// Nodes/Code Reading/Node_F_VN_ReadPharmaCodeExp2
{attribute 'linkalways'} 
{attribute 'no_explicit_call' := 'This FB is a CLASS and must be accessed using methods or properties'}
{attribute 'enable_dynamic_creation'}
FUNCTION_BLOCK Node_F_VN_ReadPharmaCodeExp2 EXTENDS VisionNode
VAR
    ipSrcImage : _ITcVnImage;
    ipDecodedData : _ITcVnContainer;
	ipContours : _ITcVnContainer;
	nCodeNumber : _DINT(1);
	nMinBarNumber : _INT(4);
	ipAngles : _ITcVnContainer;
    hrPrev : _HRESULT(S_OK);
	hresult : _HRESULT(S_OK);
END_VAR

METHOD FB_init : BOOL
VAR_INPUT
	bInitRetains : BOOL; // if TRUE, the retain variables are initialized (warm start / cold start)
	bInCopyCode : BOOL;  // if TRUE, the instance afterwards gets moved into the copy code (online change)
END_VAR
AddInput('ipSrcImage', ipSrcImage);
AddInput('hrPrev', hrPrev);
AddParameter('nCodeNumber',nCodeNumber);
AddParameter('nMinBarNumber',nMinBarNumber);
AddOutput('ipDecodedData', ipDecodedData);
AddOutput('ipContours', ipDecodedData);
AddOutput('ipAngles', ipAngles);
AddOutput('hresult',hresult);
END_METHOD

METHOD PUBLIC  Clone : I_Node
VAR
	pNode : POINTER TO Node_F_VN_ReadPharmaCodeExp2;
END_VAR
pNode := __NEW(Node_F_VN_ReadPharmaCodeExp2);
Clone := pNode^;
END_METHOD

METHOD PROTECTED OnExecute
hresult.Value := F_VN_ReadPharmaCodeExp2(
	ipSrcImage := ipSrcImage.Value,
    ipDecodedData := ipDecodedData.Value,
	ipContours := ipContours.Value,
	nCodeNumber := nCodeNumber.Value,
	nMinBarNumber := nMinBarNumber.Value,
	ipAngles := ipAngles.Value,
	hrPrev:= hrPrev.Value);
END_METHOD

METHOD PUBLIC PreExecutionCheck
VAR_INPUT
	Check : I_PreExecutionChecks;
END_VAR
Check.IsTrue(ipSrcImage.IsValid, 'ipSrcImage must contain an image');
Check.IsTrue((ipSrcImage.HasChannelCount(1) OR ipSrcImage.HasChannelCount(3)), 'ipSrcImage must have 1 or 3 channels');

IF (ipSrcImage.HasChannelCount(1)) THEN
    Check.IsTrue(ipSrcImage.IsPixelDepth(8), 'ipSrcImage must have 8 bit pixel depth');
END_IF

IF (ipSrcImage.HasChannelCount(3)) THEN
    Check.IsTrue((ipSrcImage.IsPixelDepth(8) OR 
                 ipSrcImage.IsPixelDepth(16) OR
                 ipSrcImage.IsPixelDepth(32)), 'ipSrcImage must have 8, 16 or 32 bit pixel depth');
END_IF

Check.IsTrue((nCodeNumber.Value = 1), 'nCodeNumber, currently only 1 supported');
END_METHOD

END_FUNCTION_BLOCK

// Nodes/Code Reading/Node_F_VN_ReadQRCode
{attribute 'linkalways'} 
{attribute 'no_explicit_call' := 'This FB is a CLASS and must be accessed using methods or properties'}
{attribute 'enable_dynamic_creation'}
FUNCTION_BLOCK Node_F_VN_ReadQRCode EXTENDS VisionNode
VAR
    ipSrcImage : _ITcVnImage;
    ipDecodedData : _ITcVnContainer;
    hrPrev : _HRESULT(S_OK);
	hresult : _HRESULT(S_OK);
END_VAR

METHOD FB_init : BOOL
VAR_INPUT
	bInitRetains : BOOL; // if TRUE, the retain variables are initialized (warm start / cold start)
	bInCopyCode : BOOL;  // if TRUE, the instance afterwards gets moved into the copy code (online change)
END_VAR
AddInput('ipSrcImage', ipSrcImage);
AddInput('hrPrev', hrPrev);
AddOutput('ipDecodedData', ipDecodedData);
AddOutput('hresult',hresult);
END_METHOD

METHOD PUBLIC  Clone : I_Node
VAR
	pNode : POINTER TO Node_F_VN_ReadQRCode;
END_VAR
pNode := __NEW(Node_F_VN_ReadQRCode);
Clone := pNode^;
END_METHOD

METHOD PROTECTED OnExecute
hresult.Value := F_VN_ReadQRCode(
	ipSrcImage := ipSrcImage.Value,
    ipDecodedData := ipDecodedData.Value,
	hrPrev:= hrPrev.Value);
END_METHOD

METHOD PUBLIC PreExecutionCheck
VAR_INPUT
	Check : I_PreExecutionChecks;
END_VAR
Check.IsTrue(ipSrcImage.IsValid, 'ipSrcImage must contain an image');
Check.IsTrue((ipSrcImage.HasChannelCount(1) OR ipSrcImage.HasChannelCount(3)), 'ipSrcImage must have 1 or 3 channels');
Check.IsTrue(ipSrcImage.IsPixelDepth(8), 'ipSrcImage must have 8 bit pixel depth');
END_METHOD

END_FUNCTION_BLOCK

// Nodes/Code Reading/Node_F_VN_ReadQRCodeExp
{attribute 'linkalways'} 
{attribute 'no_explicit_call' := 'This FB is a CLASS and must be accessed using methods or properties'}
{attribute 'enable_dynamic_creation'}
FUNCTION_BLOCK Node_F_VN_ReadQRCodeExp EXTENDS VisionNode
VAR
    ipSrcImage : _ITcVnImage;
    ipDecodedData : _ITcVnContainer;
	ipContours : _ITcVnContainer;
	nCodeNumber : _DINT(1);
	eSearchStrategy : _UDINT(ETcVn2dCodeSearchStrategy.TCVN_CSS_DEFAULT);
    hrPrev : _HRESULT(S_OK);
	hresult : _HRESULT(S_OK);
END_VAR

METHOD FB_init : BOOL
VAR_INPUT
	bInitRetains : BOOL; // if TRUE, the retain variables are initialized (warm start / cold start)
	bInCopyCode : BOOL;  // if TRUE, the instance afterwards gets moved into the copy code (online change)
END_VAR
AddInput('ipSrcImage', ipSrcImage);
AddInput('hrPrev', hrPrev);
AddParameter('nCodeNumber',nCodeNumber);
AddParameter('eSearchStrategy',eSearchStrategy);
AddOutput('ipDecodedData', ipDecodedData);
AddOutput('ipContours', ipContours);
AddOutput('hresult',hresult);
END_METHOD

METHOD PUBLIC  Clone : I_Node
VAR
	pNode : POINTER TO Node_F_VN_ReadQRCodeExp;
END_VAR
pNode := __NEW(Node_F_VN_ReadQRCodeExp);
Clone := pNode^;
END_METHOD

METHOD PROTECTED OnExecute
hresult.Value := F_VN_ReadQRCodeExp(
	ipSrcImage := ipSrcImage.Value,
    ipDecodedData := ipDecodedData.Value,
	ipContours := ipContours.Value,
	nCodeNumber := nCodeNumber.Value,
	eSearchStrategy := eSearchStrategy.Value,
	hrPrev:= hrPrev.Value);
END_METHOD

METHOD PUBLIC PreExecutionCheck
VAR_INPUT
	Check : I_PreExecutionChecks;
END_VAR
Check.IsTrue(ipSrcImage.IsValid, 'ipSrcImage must contain an image');
Check.IsTrue((ipSrcImage.HasChannelCount(1) OR ipSrcImage.HasChannelCount(3)), 'ipSrcImage must have 1 or 3 channels');
Check.IsTrue(ipSrcImage.IsPixelDepth(8), 'ipSrcImage must have 8 bit pixel depth');
Check.IsTrue((nCodeNumber.Value = 1), 'nCodeNumber, currently only 1 supported');
END_METHOD

END_FUNCTION_BLOCK

// Nodes/Code Reading/Node_F_VN_ReadQRCodeExp2
{attribute 'linkalways'} 
{attribute 'no_explicit_call' := 'This FB is a CLASS and must be accessed using methods or properties'}
{attribute 'enable_dynamic_creation'}
FUNCTION_BLOCK Node_F_VN_ReadQRCodeExp2 EXTENDS VisionNode
VAR
    ipSrcImage : _ITcVnImage;
    ipDecodedData : _ITcVnContainer;
	ipContours : _ITcVnContainer;
	nCodeNumber : _DINT(1);
	eSearchStrategy : _UDINT(ETcVn2dCodeSearchStrategy.TCVN_CSS_DEFAULT);
	ipAngles : _ITcVnContainer;
    hrPrev : _HRESULT(S_OK);
	hresult : _HRESULT(S_OK);
END_VAR

METHOD FB_init : BOOL
VAR_INPUT
	bInitRetains : BOOL; // if TRUE, the retain variables are initialized (warm start / cold start)
	bInCopyCode : BOOL;  // if TRUE, the instance afterwards gets moved into the copy code (online change)
END_VAR
AddInput('ipSrcImage', ipSrcImage);
AddInput('hrPrev', hrPrev);
AddParameter('nCodeNumber',nCodeNumber);
AddParameter('eSearchStrategy',eSearchStrategy);
AddOutput('ipDecodedData', ipDecodedData);
AddOutput('ipContours', ipContours);
AddOutput('ipAngles', ipAngles);
AddOutput('hresult',hresult);
END_METHOD

METHOD PUBLIC  Clone : I_Node
VAR
	pNode : POINTER TO Node_F_VN_ReadQRCodeExp2;
END_VAR
pNode := __NEW(Node_F_VN_ReadQRCodeExp2);
Clone := pNode^;
END_METHOD

METHOD PROTECTED OnExecute
hresult.Value := F_VN_ReadQRCodeExp2(
	ipSrcImage := ipSrcImage.Value,
    ipDecodedData := ipDecodedData.Value,
	ipContours := ipContours.Value,
	nCodeNumber := nCodeNumber.Value,
	eSearchStrategy := eSearchStrategy.Value,
	ipAngles := ipAngles.Value,
	hrPrev:= hrPrev.Value);
END_METHOD

METHOD PUBLIC PreExecutionCheck
VAR_INPUT
	Check : I_PreExecutionChecks;
END_VAR
Check.IsTrue(ipSrcImage.IsValid, 'ipSrcImage must contain an image');
Check.IsTrue((ipSrcImage.HasChannelCount(1) OR ipSrcImage.HasChannelCount(3)), 'ipSrcImage must have 1 or 3 channels');
Check.IsTrue(ipSrcImage.IsPixelDepth(8), 'ipSrcImage must have 8 bit pixel depth');
Check.IsTrue((nCodeNumber.Value = 1), 'nCodeNumber, currently only 1 supported');
END_METHOD

END_FUNCTION_BLOCK

// Nodes/Constants/Node_ContainerType_String_SINT
{attribute 'linkalways'} 
{attribute 'no_explicit_call' := 'This FB is a CLASS and must be accessed using methods or properties'}
{attribute 'enable_dynamic_creation'}
FUNCTION_BLOCK Node_ContainerType_String_SINT EXTENDS Node
VAR
    out : _GUID;
END_VAR

METHOD FB_init : BOOL
VAR_INPUT
	bInitRetains : BOOL; // if TRUE, the retain variables are initialized (warm start / cold start)
	bInCopyCode : BOOL;  // if TRUE, the instance afterwards gets moved into the copy code (online change)
END_VAR
AddOutput('out', out);
END_METHOD

METHOD PUBLIC  Clone : I_Node
VAR
	pNode : POINTER TO Node_ContainerType_String_SINT;
END_VAR
pNode := __NEW(Node_ContainerType_String_SINT);
Clone := pNode^;
END_METHOD

METHOD PROTECTED OnExecute
out.Value := ContainerType_String_SINT;
END_METHOD

END_FUNCTION_BLOCK

// Nodes/Constants/Node_ContainerType_Vector_DINT
{attribute 'linkalways'} 
{attribute 'no_explicit_call' := 'This FB is a CLASS and must be accessed using methods or properties'}
{attribute 'enable_dynamic_creation'}
FUNCTION_BLOCK Node_ContainerType_Vector_DINT EXTENDS Node
VAR
    out : _GUID;
END_VAR

METHOD FB_init : BOOL
VAR_INPUT
	bInitRetains : BOOL; // if TRUE, the retain variables are initialized (warm start / cold start)
	bInCopyCode : BOOL;  // if TRUE, the instance afterwards gets moved into the copy code (online change)
END_VAR
AddOutput('out', out);
END_METHOD

METHOD PUBLIC  Clone : I_Node
VAR
	pNode : POINTER TO Node_ContainerType_Vector_DINT;
END_VAR
pNode := __NEW(Node_ContainerType_Vector_DINT);
Clone := pNode^;
END_METHOD

METHOD PROTECTED OnExecute
out.Value := ContainerType_Vector_DINT;
END_METHOD

END_FUNCTION_BLOCK

// Nodes/Constants/Node_ContainerType_Vector_INT
{attribute 'linkalways'} 
{attribute 'no_explicit_call' := 'This FB is a CLASS and must be accessed using methods or properties'}
{attribute 'enable_dynamic_creation'}
FUNCTION_BLOCK Node_ContainerType_Vector_INT EXTENDS Node
VAR
    out : _GUID;
END_VAR

METHOD FB_init : BOOL
VAR_INPUT
	bInitRetains : BOOL; // if TRUE, the retain variables are initialized (warm start / cold start)
	bInCopyCode : BOOL;  // if TRUE, the instance afterwards gets moved into the copy code (online change)
END_VAR
AddOutput('out', out);
END_METHOD

METHOD PUBLIC  Clone : I_Node
VAR
	pNode : POINTER TO Node_ContainerType_Vector_INT;
END_VAR
pNode := __NEW(Node_ContainerType_Vector_INT);
Clone := pNode^;
END_METHOD

METHOD PROTECTED OnExecute
out.Value := ContainerType_Vector_INT;
END_METHOD

END_FUNCTION_BLOCK

// Nodes/Constants/Node_ContainerType_Vector_ITcVnImage
{attribute 'linkalways'} 
{attribute 'no_explicit_call' := 'This FB is a CLASS and must be accessed using methods or properties'}
{attribute 'enable_dynamic_creation'}
FUNCTION_BLOCK Node_ContainerType_Vector_ITcVnImage EXTENDS Node
VAR
    out : _GUID;
END_VAR

METHOD FB_init : BOOL
VAR_INPUT
	bInitRetains : BOOL; // if TRUE, the retain variables are initialized (warm start / cold start)
	bInCopyCode : BOOL;  // if TRUE, the instance afterwards gets moved into the copy code (online change)
END_VAR
AddOutput('out', out);
END_METHOD

METHOD PUBLIC  Clone : I_Node
VAR
	pNode : POINTER TO Node_ContainerType_Vector_ITcVnImage;
END_VAR
pNode := __NEW(Node_ContainerType_Vector_ITcVnImage);
Clone := pNode^;
END_METHOD

METHOD PROTECTED OnExecute
out.Value := ContainerType_Vector_ITcVnImage;
END_METHOD

END_FUNCTION_BLOCK

// Nodes/Constants/Node_ContainerType_Vector_LREAL
{attribute 'linkalways'} 
{attribute 'no_explicit_call' := 'This FB is a CLASS and must be accessed using methods or properties'}
{attribute 'enable_dynamic_creation'}
FUNCTION_BLOCK Node_ContainerType_Vector_LREAL EXTENDS Node
VAR
    out : _GUID;
END_VAR

METHOD FB_init : BOOL
VAR_INPUT
	bInitRetains : BOOL; // if TRUE, the retain variables are initialized (warm start / cold start)
	bInCopyCode : BOOL;  // if TRUE, the instance afterwards gets moved into the copy code (online change)
END_VAR
AddOutput('out', out);
END_METHOD

METHOD PUBLIC  Clone : I_Node
VAR
	pNode : POINTER TO Node_ContainerType_Vector_LREAL;
END_VAR
pNode := __NEW(Node_ContainerType_Vector_LREAL);
Clone := pNode^;
END_METHOD

METHOD PROTECTED OnExecute
out.Value := ContainerType_Vector_LREAL;
END_METHOD

END_FUNCTION_BLOCK

// Nodes/Constants/Node_ContainerType_Vector_REAL
{attribute 'linkalways'} 
{attribute 'no_explicit_call' := 'This FB is a CLASS and must be accessed using methods or properties'}
{attribute 'enable_dynamic_creation'}
FUNCTION_BLOCK Node_ContainerType_Vector_REAL EXTENDS Node
VAR
    out : _GUID;
END_VAR

METHOD FB_init : BOOL
VAR_INPUT
	bInitRetains : BOOL; // if TRUE, the retain variables are initialized (warm start / cold start)
	bInCopyCode : BOOL;  // if TRUE, the instance afterwards gets moved into the copy code (online change)
END_VAR
AddOutput('out', out);
END_METHOD

METHOD PUBLIC  Clone : I_Node
VAR
	pNode : POINTER TO Node_ContainerType_Vector_REAL;
END_VAR
pNode := __NEW(Node_ContainerType_Vector_REAL);
Clone := pNode^;
END_METHOD

METHOD PROTECTED OnExecute
out.Value := ContainerType_Vector_REAL;
END_METHOD

END_FUNCTION_BLOCK

// Nodes/Constants/Node_ContainerType_Vector_SINT
{attribute 'linkalways'} 
{attribute 'no_explicit_call' := 'This FB is a CLASS and must be accessed using methods or properties'}
{attribute 'enable_dynamic_creation'}
FUNCTION_BLOCK Node_ContainerType_Vector_SINT EXTENDS Node
VAR
    out : _GUID;
END_VAR

METHOD FB_init : BOOL
VAR_INPUT
	bInitRetains : BOOL; // if TRUE, the retain variables are initialized (warm start / cold start)
	bInCopyCode : BOOL;  // if TRUE, the instance afterwards gets moved into the copy code (online change)
END_VAR
AddOutput('out', out);
END_METHOD

METHOD PUBLIC  Clone : I_Node
VAR
	pNode : POINTER TO Node_ContainerType_Vector_SINT;
END_VAR
pNode := __NEW(Node_ContainerType_Vector_SINT);
Clone := pNode^;
END_METHOD

METHOD PROTECTED OnExecute
out.Value := ContainerType_Vector_SINT;
END_METHOD

END_FUNCTION_BLOCK

// Nodes/Constants/Node_ContainerType_Vector_String_SINT
{attribute 'linkalways'} 
{attribute 'no_explicit_call' := 'This FB is a CLASS and must be accessed using methods or properties'}
{attribute 'enable_dynamic_creation'}
FUNCTION_BLOCK Node_ContainerType_Vector_String_SINT EXTENDS Node
VAR
    out : _GUID;
END_VAR

METHOD FB_init : BOOL
VAR_INPUT
	bInitRetains : BOOL; // if TRUE, the retain variables are initialized (warm start / cold start)
	bInCopyCode : BOOL;  // if TRUE, the instance afterwards gets moved into the copy code (online change)
END_VAR
AddOutput('out', out);
END_METHOD

METHOD PUBLIC  Clone : I_Node
VAR
	pNode : POINTER TO Node_ContainerType_Vector_String_SINT;
END_VAR
pNode := __NEW(Node_ContainerType_Vector_String_SINT);
Clone := pNode^;
END_METHOD

METHOD PROTECTED OnExecute
out.Value := ContainerType_Vector_String_SINT;
END_METHOD

END_FUNCTION_BLOCK

// Nodes/Constants/Node_ContainerType_Vector_TcVnDMatch
{attribute 'linkalways'} 
{attribute 'no_explicit_call' := 'This FB is a CLASS and must be accessed using methods or properties'}
{attribute 'enable_dynamic_creation'}
FUNCTION_BLOCK Node_ContainerType_Vector_TcVnDMatch EXTENDS Node
VAR
    out : _GUID;
END_VAR

METHOD FB_init : BOOL
VAR_INPUT
	bInitRetains : BOOL; // if TRUE, the retain variables are initialized (warm start / cold start)
	bInCopyCode : BOOL;  // if TRUE, the instance afterwards gets moved into the copy code (online change)
END_VAR
AddOutput('out', out);
END_METHOD

METHOD PUBLIC  Clone : I_Node
VAR
	pNode : POINTER TO Node_ContainerType_Vector_TcVnDMatch;
END_VAR
pNode := __NEW(Node_ContainerType_Vector_TcVnDMatch);
Clone := pNode^;
END_METHOD

METHOD PROTECTED OnExecute
out.Value := ContainerType_Vector_TcVnDMatch;
END_METHOD

END_FUNCTION_BLOCK

// Nodes/Constants/Node_ContainerType_Vector_TcVnKeyPoint
{attribute 'linkalways'} 
{attribute 'no_explicit_call' := 'This FB is a CLASS and must be accessed using methods or properties'}
{attribute 'enable_dynamic_creation'}
FUNCTION_BLOCK Node_ContainerType_Vector_TcVnKeyPoint EXTENDS Node
VAR
    out : _GUID;
END_VAR

METHOD FB_init : BOOL
VAR_INPUT
	bInitRetains : BOOL; // if TRUE, the retain variables are initialized (warm start / cold start)
	bInCopyCode : BOOL;  // if TRUE, the instance afterwards gets moved into the copy code (online change)
END_VAR
AddOutput('out', out);
END_METHOD

METHOD PUBLIC  Clone : I_Node
VAR
	pNode : POINTER TO Node_ContainerType_Vector_TcVnKeyPoint;
END_VAR
pNode := __NEW(Node_ContainerType_Vector_TcVnKeyPoint);
Clone := pNode^;
END_METHOD

METHOD PROTECTED OnExecute
out.Value := ContainerType_Vector_TcVnKeyPoint;
END_METHOD

END_FUNCTION_BLOCK

// Nodes/Constants/Node_ContainerType_Vector_TcVnPoint2_DINT
{attribute 'linkalways'} 
{attribute 'no_explicit_call' := 'This FB is a CLASS and must be accessed using methods or properties'}
{attribute 'enable_dynamic_creation'}
FUNCTION_BLOCK Node_ContainerType_Vector_TcVnPoint2_DINT EXTENDS Node
VAR
    out : _GUID;
END_VAR

METHOD FB_init : BOOL
VAR_INPUT
	bInitRetains : BOOL; // if TRUE, the retain variables are initialized (warm start / cold start)
	bInCopyCode : BOOL;  // if TRUE, the instance afterwards gets moved into the copy code (online change)
END_VAR
AddOutput('out', out);
END_METHOD

METHOD PUBLIC  Clone : I_Node
VAR
	pNode : POINTER TO Node_ContainerType_Vector_TcVnPoint2_DINT;
END_VAR
pNode := __NEW(Node_ContainerType_Vector_TcVnPoint2_DINT);
Clone := pNode^;
END_METHOD

METHOD PROTECTED OnExecute
out.Value := ContainerType_Vector_TcVnPoint2_DINT;
END_METHOD

END_FUNCTION_BLOCK

// Nodes/Constants/Node_ContainerType_Vector_TcVnPoint2_LREAL
{attribute 'linkalways'} 
{attribute 'no_explicit_call' := 'This FB is a CLASS and must be accessed using methods or properties'}
{attribute 'enable_dynamic_creation'}
FUNCTION_BLOCK Node_ContainerType_Vector_TcVnPoint2_LREAL EXTENDS Node
VAR
    out : _GUID;
END_VAR

METHOD FB_init : BOOL
VAR_INPUT
	bInitRetains : BOOL; // if TRUE, the retain variables are initialized (warm start / cold start)
	bInCopyCode : BOOL;  // if TRUE, the instance afterwards gets moved into the copy code (online change)
END_VAR
AddOutput('out', out);
END_METHOD

METHOD PUBLIC  Clone : I_Node
VAR
	pNode : POINTER TO Node_ContainerType_Vector_TcVnPoint2_LREAL;
END_VAR
pNode := __NEW(Node_ContainerType_Vector_TcVnPoint2_LREAL);
Clone := pNode^;
END_METHOD

METHOD PROTECTED OnExecute
out.Value := ContainerType_Vector_TcVnPoint2_LREAL;
END_METHOD

END_FUNCTION_BLOCK

// Nodes/Constants/Node_ContainerType_Vector_TcVnPoint2_REAL
{attribute 'linkalways'} 
{attribute 'no_explicit_call' := 'This FB is a CLASS and must be accessed using methods or properties'}
{attribute 'enable_dynamic_creation'}
FUNCTION_BLOCK Node_ContainerType_Vector_TcVnPoint2_REAL EXTENDS Node
VAR
    out : _GUID;
END_VAR

METHOD FB_init : BOOL
VAR_INPUT
	bInitRetains : BOOL; // if TRUE, the retain variables are initialized (warm start / cold start)
	bInCopyCode : BOOL;  // if TRUE, the instance afterwards gets moved into the copy code (online change)
END_VAR
AddOutput('out', out);
END_METHOD

METHOD PUBLIC  Clone : I_Node
VAR
	pNode : POINTER TO Node_ContainerType_Vector_TcVnPoint2_REAL;
END_VAR
pNode := __NEW(Node_ContainerType_Vector_TcVnPoint2_REAL);
Clone := pNode^;
END_METHOD

METHOD PROTECTED OnExecute
out.Value := ContainerType_Vector_TcVnPoint2_REAL;
END_METHOD

END_FUNCTION_BLOCK

// Nodes/Constants/Node_ContainerType_Vector_TcVnPoint3_LREAL
{attribute 'linkalways'} 
{attribute 'no_explicit_call' := 'This FB is a CLASS and must be accessed using methods or properties'}
{attribute 'enable_dynamic_creation'}
FUNCTION_BLOCK Node_ContainerType_Vector_TcVnPoint3_LREAL EXTENDS Node
VAR
    out : _GUID;
END_VAR

METHOD FB_init : BOOL
VAR_INPUT
	bInitRetains : BOOL; // if TRUE, the retain variables are initialized (warm start / cold start)
	bInCopyCode : BOOL;  // if TRUE, the instance afterwards gets moved into the copy code (online change)
END_VAR
AddOutput('out', out);
END_METHOD

METHOD PUBLIC  Clone : I_Node
VAR
	pNode : POINTER TO Node_ContainerType_Vector_TcVnPoint3_LREAL;
END_VAR
pNode := __NEW(Node_ContainerType_Vector_TcVnPoint3_LREAL);
Clone := pNode^;
END_METHOD

METHOD PROTECTED OnExecute
out.Value := ContainerType_Vector_TcVnPoint3_LREAL;
END_METHOD

END_FUNCTION_BLOCK

// Nodes/Constants/Node_ContainerType_Vector_TcVnPoint3_REAL
{attribute 'linkalways'} 
{attribute 'no_explicit_call' := 'This FB is a CLASS and must be accessed using methods or properties'}
{attribute 'enable_dynamic_creation'}
FUNCTION_BLOCK Node_ContainerType_Vector_TcVnPoint3_REAL EXTENDS Node
VAR
    out : _GUID;
END_VAR

METHOD FB_init : BOOL
VAR_INPUT
	bInitRetains : BOOL; // if TRUE, the retain variables are initialized (warm start / cold start)
	bInCopyCode : BOOL;  // if TRUE, the instance afterwards gets moved into the copy code (online change)
END_VAR
AddOutput('out', out);
END_METHOD

METHOD PUBLIC  Clone : I_Node
VAR
	pNode : POINTER TO Node_ContainerType_Vector_TcVnPoint3_REAL;
END_VAR
pNode := __NEW(Node_ContainerType_Vector_TcVnPoint3_REAL);
Clone := pNode^;
END_METHOD

METHOD PROTECTED OnExecute
out.Value := ContainerType_Vector_TcVnPoint3_REAL;
END_METHOD

END_FUNCTION_BLOCK

// Nodes/Constants/Node_ContainerType_Vector_TcVnRectangle_DINT
{attribute 'linkalways'} 
{attribute 'no_explicit_call' := 'This FB is a CLASS and must be accessed using methods or properties'}
{attribute 'enable_dynamic_creation'}
FUNCTION_BLOCK Node_ContainerType_Vector_TcVnRectangle_DINT EXTENDS Node
VAR
    out : _GUID;
END_VAR

METHOD FB_init : BOOL
VAR_INPUT
	bInitRetains : BOOL; // if TRUE, the retain variables are initialized (warm start / cold start)
	bInCopyCode : BOOL;  // if TRUE, the instance afterwards gets moved into the copy code (online change)
END_VAR
AddOutput('out', out);
END_METHOD

METHOD PUBLIC  Clone : I_Node
VAR
	pNode : POINTER TO Node_ContainerType_Vector_TcVnRectangle_DINT;
END_VAR
pNode := __NEW(Node_ContainerType_Vector_TcVnRectangle_DINT);
Clone := pNode^;
END_METHOD

METHOD PROTECTED OnExecute
out.Value := ContainerType_Vector_TcVnRectangle_DINT;
END_METHOD

END_FUNCTION_BLOCK

// Nodes/Constants/Node_ContainerType_Vector_TcVnRotatedRectangle
{attribute 'linkalways'} 
{attribute 'no_explicit_call' := 'This FB is a CLASS and must be accessed using methods or properties'}
{attribute 'enable_dynamic_creation'}
FUNCTION_BLOCK Node_ContainerType_Vector_TcVnRotatedRectangle EXTENDS Node
VAR
    out : _GUID;
END_VAR

METHOD FB_init : BOOL
VAR_INPUT
	bInitRetains : BOOL; // if TRUE, the retain variables are initialized (warm start / cold start)
	bInCopyCode : BOOL;  // if TRUE, the instance afterwards gets moved into the copy code (online change)
END_VAR
AddOutput('out', out);
END_METHOD

METHOD PUBLIC  Clone : I_Node
VAR
	pNode : POINTER TO Node_ContainerType_Vector_TcVnRotatedRectangle;
END_VAR
pNode := __NEW(Node_ContainerType_Vector_TcVnRotatedRectangle);
Clone := pNode^;
END_METHOD

METHOD PROTECTED OnExecute
out.Value := ContainerType_Vector_TcVnRotatedRectangle;
END_METHOD

END_FUNCTION_BLOCK

// Nodes/Constants/Node_ContainerType_Vector_TcVnVector2_DINT
{attribute 'linkalways'} 
{attribute 'no_explicit_call' := 'This FB is a CLASS and must be accessed using methods or properties'}
{attribute 'enable_dynamic_creation'}
FUNCTION_BLOCK Node_ContainerType_Vector_TcVnVector2_DINT EXTENDS Node
VAR
    out : _GUID;
END_VAR

METHOD FB_init : BOOL
VAR_INPUT
	bInitRetains : BOOL; // if TRUE, the retain variables are initialized (warm start / cold start)
	bInCopyCode : BOOL;  // if TRUE, the instance afterwards gets moved into the copy code (online change)
END_VAR
AddOutput('out', out);
END_METHOD

METHOD PUBLIC  Clone : I_Node
VAR
	pNode : POINTER TO Node_ContainerType_Vector_TcVnVector2_DINT;
END_VAR
pNode := __NEW(Node_ContainerType_Vector_TcVnVector2_DINT);
Clone := pNode^;
END_METHOD

METHOD PROTECTED OnExecute
out.Value := ContainerType_Vector_TcVnVector2_DINT;
END_METHOD

END_FUNCTION_BLOCK

// Nodes/Constants/Node_ContainerType_Vector_TcVnVector2_INT
{attribute 'linkalways'} 
{attribute 'no_explicit_call' := 'This FB is a CLASS and must be accessed using methods or properties'}
{attribute 'enable_dynamic_creation'}
FUNCTION_BLOCK Node_ContainerType_Vector_TcVnVector2_INT EXTENDS Node
VAR
    out : _GUID;
END_VAR

METHOD FB_init : BOOL
VAR_INPUT
	bInitRetains : BOOL; // if TRUE, the retain variables are initialized (warm start / cold start)
	bInCopyCode : BOOL;  // if TRUE, the instance afterwards gets moved into the copy code (online change)
END_VAR
AddOutput('out', out);
END_METHOD

METHOD PUBLIC  Clone : I_Node
VAR
	pNode : POINTER TO Node_ContainerType_Vector_TcVnVector2_INT;
END_VAR
pNode := __NEW(Node_ContainerType_Vector_TcVnVector2_INT);
Clone := pNode^;
END_METHOD

METHOD PROTECTED OnExecute
out.Value := ContainerType_Vector_TcVnVector2_INT;
END_METHOD

END_FUNCTION_BLOCK

// Nodes/Constants/Node_ContainerType_Vector_TcVnVector2_REAL
{attribute 'linkalways'} 
{attribute 'no_explicit_call' := 'This FB is a CLASS and must be accessed using methods or properties'}
{attribute 'enable_dynamic_creation'}
FUNCTION_BLOCK Node_ContainerType_Vector_TcVnVector2_REAL EXTENDS Node
VAR
    out : _GUID;
END_VAR

METHOD FB_init : BOOL
VAR_INPUT
	bInitRetains : BOOL; // if TRUE, the retain variables are initialized (warm start / cold start)
	bInCopyCode : BOOL;  // if TRUE, the instance afterwards gets moved into the copy code (online change)
END_VAR
AddOutput('out', out);
END_METHOD

METHOD PUBLIC  Clone : I_Node
VAR
	pNode : POINTER TO Node_ContainerType_Vector_TcVnVector2_REAL;
END_VAR
pNode := __NEW(Node_ContainerType_Vector_TcVnVector2_REAL);
Clone := pNode^;
END_METHOD

METHOD PROTECTED OnExecute
out.Value := ContainerType_Vector_TcVnVector2_REAL;
END_METHOD

END_FUNCTION_BLOCK

// Nodes/Constants/Node_ContainerType_Vector_TcVnVector2_SINT
{attribute 'linkalways'} 
{attribute 'no_explicit_call' := 'This FB is a CLASS and must be accessed using methods or properties'}
{attribute 'enable_dynamic_creation'}
FUNCTION_BLOCK Node_ContainerType_Vector_TcVnVector2_SINT EXTENDS Node
VAR
    out : _GUID;
END_VAR

METHOD FB_init : BOOL
VAR_INPUT
	bInitRetains : BOOL; // if TRUE, the retain variables are initialized (warm start / cold start)
	bInCopyCode : BOOL;  // if TRUE, the instance afterwards gets moved into the copy code (online change)
END_VAR
AddOutput('out', out);
END_METHOD

METHOD PUBLIC  Clone : I_Node
VAR
	pNode : POINTER TO Node_ContainerType_Vector_TcVnVector2_SINT;
END_VAR
pNode := __NEW(Node_ContainerType_Vector_TcVnVector2_SINT);
Clone := pNode^;
END_METHOD

METHOD PROTECTED OnExecute
out.Value := ContainerType_Vector_TcVnVector2_SINT;
END_METHOD

END_FUNCTION_BLOCK

// Nodes/Constants/Node_ContainerType_Vector_TcVnVector2_UINT
{attribute 'linkalways'} 
{attribute 'no_explicit_call' := 'This FB is a CLASS and must be accessed using methods or properties'}
{attribute 'enable_dynamic_creation'}
FUNCTION_BLOCK Node_ContainerType_Vector_TcVnVector2_UINT EXTENDS Node
VAR
    out : _GUID;
END_VAR

METHOD FB_init : BOOL
VAR_INPUT
	bInitRetains : BOOL; // if TRUE, the retain variables are initialized (warm start / cold start)
	bInCopyCode : BOOL;  // if TRUE, the instance afterwards gets moved into the copy code (online change)
END_VAR
AddOutput('out', out);
END_METHOD

METHOD PUBLIC  Clone : I_Node
VAR
	pNode : POINTER TO Node_ContainerType_Vector_TcVnVector2_UINT;
END_VAR
pNode := __NEW(Node_ContainerType_Vector_TcVnVector2_UINT);
Clone := pNode^;
END_METHOD

METHOD PROTECTED OnExecute
out.Value := ContainerType_Vector_TcVnVector2_UINT;
END_METHOD

END_FUNCTION_BLOCK

// Nodes/Constants/Node_ContainerType_Vector_TcVnVector2_USINT
{attribute 'linkalways'} 
{attribute 'no_explicit_call' := 'This FB is a CLASS and must be accessed using methods or properties'}
{attribute 'enable_dynamic_creation'}
FUNCTION_BLOCK Node_ContainerType_Vector_TcVnVector2_USINT EXTENDS Node
VAR
    out : _GUID;
END_VAR

METHOD FB_init : BOOL
VAR_INPUT
	bInitRetains : BOOL; // if TRUE, the retain variables are initialized (warm start / cold start)
	bInCopyCode : BOOL;  // if TRUE, the instance afterwards gets moved into the copy code (online change)
END_VAR
AddOutput('out', out);
END_METHOD

METHOD PUBLIC  Clone : I_Node
VAR
	pNode : POINTER TO Node_ContainerType_Vector_TcVnVector2_USINT;
END_VAR
pNode := __NEW(Node_ContainerType_Vector_TcVnVector2_USINT);
Clone := pNode^;
END_METHOD

METHOD PROTECTED OnExecute
out.Value := ContainerType_Vector_TcVnVector2_USINT;
END_METHOD

END_FUNCTION_BLOCK

// Nodes/Constants/Node_ContainerType_Vector_TcVnVector3_INT
{attribute 'linkalways'} 
{attribute 'no_explicit_call' := 'This FB is a CLASS and must be accessed using methods or properties'}
{attribute 'enable_dynamic_creation'}
FUNCTION_BLOCK Node_ContainerType_Vector_TcVnVector3_INT EXTENDS Node
VAR
    out : _GUID;
END_VAR

METHOD FB_init : BOOL
VAR_INPUT
	bInitRetains : BOOL; // if TRUE, the retain variables are initialized (warm start / cold start)
	bInCopyCode : BOOL;  // if TRUE, the instance afterwards gets moved into the copy code (online change)
END_VAR
AddOutput('out', out);
END_METHOD

METHOD PUBLIC  Clone : I_Node
VAR
	pNode : POINTER TO Node_ContainerType_Vector_TcVnVector3_INT;
END_VAR
pNode := __NEW(Node_ContainerType_Vector_TcVnVector3_INT);
Clone := pNode^;
END_METHOD

METHOD PROTECTED OnExecute
out.Value := ContainerType_Vector_TcVnVector3_INT;
END_METHOD

END_FUNCTION_BLOCK

// Nodes/Constants/Node_ContainerType_Vector_TcVnVector3_REAL
{attribute 'linkalways'} 
{attribute 'no_explicit_call' := 'This FB is a CLASS and must be accessed using methods or properties'}
{attribute 'enable_dynamic_creation'}
FUNCTION_BLOCK Node_ContainerType_Vector_TcVnVector3_REAL EXTENDS Node
VAR
    out : _GUID;
END_VAR

METHOD FB_init : BOOL
VAR_INPUT
	bInitRetains : BOOL; // if TRUE, the retain variables are initialized (warm start / cold start)
	bInCopyCode : BOOL;  // if TRUE, the instance afterwards gets moved into the copy code (online change)
END_VAR
AddOutput('out', out);
END_METHOD

METHOD PUBLIC  Clone : I_Node
VAR
	pNode : POINTER TO Node_ContainerType_Vector_TcVnVector3_REAL;
END_VAR
pNode := __NEW(Node_ContainerType_Vector_TcVnVector3_REAL);
Clone := pNode^;
END_METHOD

METHOD PROTECTED OnExecute
out.Value := ContainerType_Vector_TcVnVector3_REAL;
END_METHOD

END_FUNCTION_BLOCK

// Nodes/Constants/Node_ContainerType_Vector_TcVnVector3_SINT
{attribute 'linkalways'} 
{attribute 'no_explicit_call' := 'This FB is a CLASS and must be accessed using methods or properties'}
{attribute 'enable_dynamic_creation'}
FUNCTION_BLOCK Node_ContainerType_Vector_TcVnVector3_SINT EXTENDS Node
VAR
    out : _GUID;
END_VAR

METHOD FB_init : BOOL
VAR_INPUT
	bInitRetains : BOOL; // if TRUE, the retain variables are initialized (warm start / cold start)
	bInCopyCode : BOOL;  // if TRUE, the instance afterwards gets moved into the copy code (online change)
END_VAR
AddOutput('out', out);
END_METHOD

METHOD PUBLIC  Clone : I_Node
VAR
	pNode : POINTER TO Node_ContainerType_Vector_TcVnVector3_SINT;
END_VAR
pNode := __NEW(Node_ContainerType_Vector_TcVnVector3_SINT);
Clone := pNode^;
END_METHOD

METHOD PROTECTED OnExecute
out.Value := ContainerType_Vector_TcVnVector3_SINT;
END_METHOD

END_FUNCTION_BLOCK

// Nodes/Constants/Node_ContainerType_Vector_TcVnVector3_UINT
{attribute 'linkalways'} 
{attribute 'no_explicit_call' := 'This FB is a CLASS and must be accessed using methods or properties'}
{attribute 'enable_dynamic_creation'}
FUNCTION_BLOCK Node_ContainerType_Vector_TcVnVector3_UINT EXTENDS Node
VAR
    out : _GUID;
END_VAR

METHOD FB_init : BOOL
VAR_INPUT
	bInitRetains : BOOL; // if TRUE, the retain variables are initialized (warm start / cold start)
	bInCopyCode : BOOL;  // if TRUE, the instance afterwards gets moved into the copy code (online change)
END_VAR
AddOutput('out', out);
END_METHOD

METHOD PUBLIC  Clone : I_Node
VAR
	pNode : POINTER TO Node_ContainerType_Vector_TcVnVector3_UINT;
END_VAR
pNode := __NEW(Node_ContainerType_Vector_TcVnVector3_UINT);
Clone := pNode^;
END_METHOD

METHOD PROTECTED OnExecute
out.Value := ContainerType_Vector_TcVnVector3_UINT;
END_METHOD

END_FUNCTION_BLOCK

// Nodes/Constants/Node_ContainerType_Vector_TcVnVector3_USINT
{attribute 'linkalways'} 
{attribute 'no_explicit_call' := 'This FB is a CLASS and must be accessed using methods or properties'}
{attribute 'enable_dynamic_creation'}
FUNCTION_BLOCK Node_ContainerType_Vector_TcVnVector3_USINT EXTENDS Node
VAR
    out : _GUID;
END_VAR

METHOD FB_init : BOOL
VAR_INPUT
	bInitRetains : BOOL; // if TRUE, the retain variables are initialized (warm start / cold start)
	bInCopyCode : BOOL;  // if TRUE, the instance afterwards gets moved into the copy code (online change)
END_VAR
AddOutput('out', out);
END_METHOD

METHOD PUBLIC  Clone : I_Node
VAR
	pNode : POINTER TO Node_ContainerType_Vector_TcVnVector3_USINT;
END_VAR
pNode := __NEW(Node_ContainerType_Vector_TcVnVector3_USINT);
Clone := pNode^;
END_METHOD

METHOD PROTECTED OnExecute
out.Value := ContainerType_Vector_TcVnVector3_USINT;
END_METHOD

END_FUNCTION_BLOCK

// Nodes/Constants/Node_ContainerType_Vector_TcVnVector4_DINT
{attribute 'linkalways'} 
{attribute 'no_explicit_call' := 'This FB is a CLASS and must be accessed using methods or properties'}
{attribute 'enable_dynamic_creation'}
FUNCTION_BLOCK Node_ContainerType_Vector_TcVnVector4_DINT EXTENDS Node
VAR
    out : _GUID;
END_VAR

METHOD FB_init : BOOL
VAR_INPUT
	bInitRetains : BOOL; // if TRUE, the retain variables are initialized (warm start / cold start)
	bInCopyCode : BOOL;  // if TRUE, the instance afterwards gets moved into the copy code (online change)
END_VAR
AddOutput('out', out);
END_METHOD

METHOD PUBLIC  Clone : I_Node
VAR
	pNode : POINTER TO Node_ContainerType_Vector_TcVnVector4_DINT;
END_VAR
pNode := __NEW(Node_ContainerType_Vector_TcVnVector4_DINT);
Clone := pNode^;
END_METHOD

METHOD PROTECTED OnExecute
out.Value := ContainerType_Vector_TcVnVector4_DINT;
END_METHOD

END_FUNCTION_BLOCK

// Nodes/Constants/Node_ContainerType_Vector_TcVnVector4_INT
{attribute 'linkalways'} 
{attribute 'no_explicit_call' := 'This FB is a CLASS and must be accessed using methods or properties'}
{attribute 'enable_dynamic_creation'}
FUNCTION_BLOCK Node_ContainerType_Vector_TcVnVector4_INT EXTENDS Node
VAR
    out : _GUID;
END_VAR

METHOD FB_init : BOOL
VAR_INPUT
	bInitRetains : BOOL; // if TRUE, the retain variables are initialized (warm start / cold start)
	bInCopyCode : BOOL;  // if TRUE, the instance afterwards gets moved into the copy code (online change)
END_VAR
AddOutput('out', out);
END_METHOD

METHOD PUBLIC  Clone : I_Node
VAR
	pNode : POINTER TO Node_ContainerType_Vector_TcVnVector4_INT;
END_VAR
pNode := __NEW(Node_ContainerType_Vector_TcVnVector4_INT);
Clone := pNode^;
END_METHOD

METHOD PROTECTED OnExecute
out.Value := ContainerType_Vector_TcVnVector4_INT;
END_METHOD

END_FUNCTION_BLOCK

// Nodes/Constants/Node_ContainerType_Vector_TcVnVector4_LREAL
{attribute 'linkalways'} 
{attribute 'no_explicit_call' := 'This FB is a CLASS and must be accessed using methods or properties'}
{attribute 'enable_dynamic_creation'}
FUNCTION_BLOCK Node_ContainerType_Vector_TcVnVector4_LREAL EXTENDS Node
VAR
    out : _GUID;
END_VAR

METHOD FB_init : BOOL
VAR_INPUT
	bInitRetains : BOOL; // if TRUE, the retain variables are initialized (warm start / cold start)
	bInCopyCode : BOOL;  // if TRUE, the instance afterwards gets moved into the copy code (online change)
END_VAR
AddOutput('out', out);
END_METHOD

METHOD PUBLIC  Clone : I_Node
VAR
	pNode : POINTER TO Node_ContainerType_Vector_TcVnVector4_LREAL;
END_VAR
pNode := __NEW(Node_ContainerType_Vector_TcVnVector4_LREAL);
Clone := pNode^;
END_METHOD

METHOD PROTECTED OnExecute
out.Value := ContainerType_Vector_TcVnVector4_LREAL;
END_METHOD

END_FUNCTION_BLOCK

// Nodes/Constants/Node_ContainerType_Vector_TcVnVector4_REAL
{attribute 'linkalways'} 
{attribute 'no_explicit_call' := 'This FB is a CLASS and must be accessed using methods or properties'}
{attribute 'enable_dynamic_creation'}
FUNCTION_BLOCK Node_ContainerType_Vector_TcVnVector4_REAL EXTENDS Node
VAR
    out : _GUID;
END_VAR

METHOD FB_init : BOOL
VAR_INPUT
	bInitRetains : BOOL; // if TRUE, the retain variables are initialized (warm start / cold start)
	bInCopyCode : BOOL;  // if TRUE, the instance afterwards gets moved into the copy code (online change)
END_VAR
AddOutput('out', out);
END_METHOD

METHOD PUBLIC  Clone : I_Node
VAR
	pNode : POINTER TO Node_ContainerType_Vector_TcVnVector4_REAL;
END_VAR
pNode := __NEW(Node_ContainerType_Vector_TcVnVector4_REAL);
Clone := pNode^;
END_METHOD

METHOD PROTECTED OnExecute
out.Value := ContainerType_Vector_TcVnVector4_REAL;
END_METHOD

END_FUNCTION_BLOCK

// Nodes/Constants/Node_ContainerType_Vector_TcVnVector4_SINT
{attribute 'linkalways'} 
{attribute 'no_explicit_call' := 'This FB is a CLASS and must be accessed using methods or properties'}
{attribute 'enable_dynamic_creation'}
FUNCTION_BLOCK Node_ContainerType_Vector_TcVnVector4_SINT EXTENDS Node
VAR
    out : _GUID;
END_VAR

METHOD FB_init : BOOL
VAR_INPUT
	bInitRetains : BOOL; // if TRUE, the retain variables are initialized (warm start / cold start)
	bInCopyCode : BOOL;  // if TRUE, the instance afterwards gets moved into the copy code (online change)
END_VAR
AddOutput('out', out);
END_METHOD

METHOD PUBLIC  Clone : I_Node
VAR
	pNode : POINTER TO Node_ContainerType_Vector_TcVnVector4_SINT;
END_VAR
pNode := __NEW(Node_ContainerType_Vector_TcVnVector4_SINT);
Clone := pNode^;
END_METHOD

METHOD PROTECTED OnExecute
out.Value := ContainerType_Vector_TcVnVector4_SINT;
END_METHOD

END_FUNCTION_BLOCK

// Nodes/Constants/Node_ContainerType_Vector_TcVnVector4_UINT
{attribute 'linkalways'} 
{attribute 'no_explicit_call' := 'This FB is a CLASS and must be accessed using methods or properties'}
{attribute 'enable_dynamic_creation'}
FUNCTION_BLOCK Node_ContainerType_Vector_TcVnVector4_UINT EXTENDS Node
VAR
    out : _GUID;
END_VAR

METHOD FB_init : BOOL
VAR_INPUT
	bInitRetains : BOOL; // if TRUE, the retain variables are initialized (warm start / cold start)
	bInCopyCode : BOOL;  // if TRUE, the instance afterwards gets moved into the copy code (online change)
END_VAR
AddOutput('out', out);
END_METHOD

METHOD PUBLIC  Clone : I_Node
VAR
	pNode : POINTER TO Node_ContainerType_Vector_TcVnVector4_UINT;
END_VAR
pNode := __NEW(Node_ContainerType_Vector_TcVnVector4_UINT);
Clone := pNode^;
END_METHOD

METHOD PROTECTED OnExecute
out.Value := ContainerType_Vector_TcVnVector4_UINT;
END_METHOD

END_FUNCTION_BLOCK

// Nodes/Constants/Node_ContainerType_Vector_TcVnVector4_USINT
{attribute 'linkalways'} 
{attribute 'no_explicit_call' := 'This FB is a CLASS and must be accessed using methods or properties'}
{attribute 'enable_dynamic_creation'}
FUNCTION_BLOCK Node_ContainerType_Vector_TcVnVector4_USINT EXTENDS Node
VAR
    out : _GUID;
END_VAR

METHOD FB_init : BOOL
VAR_INPUT
	bInitRetains : BOOL; // if TRUE, the retain variables are initialized (warm start / cold start)
	bInCopyCode : BOOL;  // if TRUE, the instance afterwards gets moved into the copy code (online change)
END_VAR
AddOutput('out', out);
END_METHOD

METHOD PUBLIC  Clone : I_Node
VAR
	pNode : POINTER TO Node_ContainerType_Vector_TcVnVector4_USINT;
END_VAR
pNode := __NEW(Node_ContainerType_Vector_TcVnVector4_USINT);
Clone := pNode^;
END_METHOD

METHOD PROTECTED OnExecute
out.Value := ContainerType_Vector_TcVnVector4_USINT;
END_METHOD

END_FUNCTION_BLOCK

// Nodes/Constants/Node_ContainerType_Vector_UDINT
{attribute 'linkalways'} 
{attribute 'no_explicit_call' := 'This FB is a CLASS and must be accessed using methods or properties'}
{attribute 'enable_dynamic_creation'}
FUNCTION_BLOCK Node_ContainerType_Vector_UDINT EXTENDS Node
VAR
    out : _GUID;
END_VAR

METHOD FB_init : BOOL
VAR_INPUT
	bInitRetains : BOOL; // if TRUE, the retain variables are initialized (warm start / cold start)
	bInCopyCode : BOOL;  // if TRUE, the instance afterwards gets moved into the copy code (online change)
END_VAR
AddOutput('out', out);
END_METHOD

METHOD PUBLIC  Clone : I_Node
VAR
	pNode : POINTER TO Node_ContainerType_Vector_UDINT;
END_VAR
pNode := __NEW(Node_ContainerType_Vector_UDINT);
Clone := pNode^;
END_METHOD

METHOD PROTECTED OnExecute
out.Value := ContainerType_Vector_UDINT;
END_METHOD

END_FUNCTION_BLOCK

// Nodes/Constants/Node_ContainerType_Vector_UINT
{attribute 'linkalways'} 
{attribute 'no_explicit_call' := 'This FB is a CLASS and must be accessed using methods or properties'}
{attribute 'enable_dynamic_creation'}
FUNCTION_BLOCK Node_ContainerType_Vector_UINT EXTENDS Node
VAR
    out : _GUID;
END_VAR

METHOD FB_init : BOOL
VAR_INPUT
	bInitRetains : BOOL; // if TRUE, the retain variables are initialized (warm start / cold start)
	bInCopyCode : BOOL;  // if TRUE, the instance afterwards gets moved into the copy code (online change)
END_VAR
AddOutput('out', out);
END_METHOD

METHOD PUBLIC  Clone : I_Node
VAR
	pNode : POINTER TO Node_ContainerType_Vector_UINT;
END_VAR
pNode := __NEW(Node_ContainerType_Vector_UINT);
Clone := pNode^;
END_METHOD

METHOD PROTECTED OnExecute
out.Value := ContainerType_Vector_UINT;
END_METHOD

END_FUNCTION_BLOCK

// Nodes/Constants/Node_ContainerType_Vector_ULINT
{attribute 'linkalways'} 
{attribute 'no_explicit_call' := 'This FB is a CLASS and must be accessed using methods or properties'}
{attribute 'enable_dynamic_creation'}
FUNCTION_BLOCK Node_ContainerType_Vector_ULINT EXTENDS Node
VAR
    out : _GUID;
END_VAR

METHOD FB_init : BOOL
VAR_INPUT
	bInitRetains : BOOL; // if TRUE, the retain variables are initialized (warm start / cold start)
	bInCopyCode : BOOL;  // if TRUE, the instance afterwards gets moved into the copy code (online change)
END_VAR
AddOutput('out', out);
END_METHOD

METHOD PUBLIC  Clone : I_Node
VAR
	pNode : POINTER TO Node_ContainerType_Vector_ULINT;
END_VAR
pNode := __NEW(Node_ContainerType_Vector_ULINT);
Clone := pNode^;
END_METHOD

METHOD PROTECTED OnExecute
out.Value := ContainerType_Vector_ULINT;
END_METHOD

END_FUNCTION_BLOCK

// Nodes/Constants/Node_ContainerType_Vector_USINT
{attribute 'linkalways'} 
{attribute 'no_explicit_call' := 'This FB is a CLASS and must be accessed using methods or properties'}
{attribute 'enable_dynamic_creation'}
FUNCTION_BLOCK Node_ContainerType_Vector_USINT EXTENDS Node
VAR
    out : _GUID;
END_VAR

METHOD FB_init : BOOL
VAR_INPUT
	bInitRetains : BOOL; // if TRUE, the retain variables are initialized (warm start / cold start)
	bInCopyCode : BOOL;  // if TRUE, the instance afterwards gets moved into the copy code (online change)
END_VAR
AddOutput('out', out);
END_METHOD

METHOD PUBLIC  Clone : I_Node
VAR
	pNode : POINTER TO Node_ContainerType_Vector_USINT;
END_VAR
pNode := __NEW(Node_ContainerType_Vector_USINT);
Clone := pNode^;
END_METHOD

METHOD PROTECTED OnExecute
out.Value := ContainerType_Vector_USINT;
END_METHOD

END_FUNCTION_BLOCK

// Nodes/Constants/Node_ContainerType_Vector_Vector_LREAL
{attribute 'linkalways'} 
{attribute 'no_explicit_call' := 'This FB is a CLASS and must be accessed using methods or properties'}
{attribute 'enable_dynamic_creation'}
FUNCTION_BLOCK Node_ContainerType_Vector_Vector_LREAL EXTENDS Node
VAR
    out : _GUID;
END_VAR

METHOD FB_init : BOOL
VAR_INPUT
	bInitRetains : BOOL; // if TRUE, the retain variables are initialized (warm start / cold start)
	bInCopyCode : BOOL;  // if TRUE, the instance afterwards gets moved into the copy code (online change)
END_VAR
AddOutput('out', out);
END_METHOD

METHOD PUBLIC  Clone : I_Node
VAR
	pNode : POINTER TO Node_ContainerType_Vector_Vector_LREAL;
END_VAR
pNode := __NEW(Node_ContainerType_Vector_Vector_LREAL);
Clone := pNode^;
END_METHOD

METHOD PROTECTED OnExecute
out.Value := ContainerType_Vector_Vector_LREAL;
END_METHOD

END_FUNCTION_BLOCK

// Nodes/Constants/Node_ContainerType_Vector_Vector_REAL
{attribute 'linkalways'} 
{attribute 'no_explicit_call' := 'This FB is a CLASS and must be accessed using methods or properties'}
{attribute 'enable_dynamic_creation'}
FUNCTION_BLOCK Node_ContainerType_Vector_Vector_REAL EXTENDS Node
VAR
    out : _GUID;
END_VAR

METHOD FB_init : BOOL
VAR_INPUT
	bInitRetains : BOOL; // if TRUE, the retain variables are initialized (warm start / cold start)
	bInCopyCode : BOOL;  // if TRUE, the instance afterwards gets moved into the copy code (online change)
END_VAR
AddOutput('out', out);
END_METHOD

METHOD PUBLIC  Clone : I_Node
VAR
	pNode : POINTER TO Node_ContainerType_Vector_Vector_REAL;
END_VAR
pNode := __NEW(Node_ContainerType_Vector_Vector_REAL);
Clone := pNode^;
END_METHOD

METHOD PROTECTED OnExecute
out.Value := ContainerType_Vector_Vector_REAL;
END_METHOD

END_FUNCTION_BLOCK

// Nodes/Constants/Node_ContainerType_Vector_Vector_TcVnDMatch
{attribute 'linkalways'} 
{attribute 'no_explicit_call' := 'This FB is a CLASS and must be accessed using methods or properties'}
{attribute 'enable_dynamic_creation'}
FUNCTION_BLOCK Node_ContainerType_Vector_Vector_TcVnDMatch EXTENDS Node
VAR
    out : _GUID;
END_VAR

METHOD FB_init : BOOL
VAR_INPUT
	bInitRetains : BOOL; // if TRUE, the retain variables are initialized (warm start / cold start)
	bInCopyCode : BOOL;  // if TRUE, the instance afterwards gets moved into the copy code (online change)
END_VAR
AddOutput('out', out);
END_METHOD

METHOD PUBLIC  Clone : I_Node
VAR
	pNode : POINTER TO Node_ContainerType_Vector_Vector_TcVnDMatch;
END_VAR
pNode := __NEW(Node_ContainerType_Vector_Vector_TcVnDMatch);
Clone := pNode^;
END_METHOD

METHOD PROTECTED OnExecute
out.Value := ContainerType_Vector_Vector_TcVnDMatch;
END_METHOD

END_FUNCTION_BLOCK

// Nodes/Constants/Node_ContainerType_Vector_Vector_TcVnPoint2_DINT
{attribute 'linkalways'} 
{attribute 'no_explicit_call' := 'This FB is a CLASS and must be accessed using methods or properties'}
{attribute 'enable_dynamic_creation'}
FUNCTION_BLOCK Node_ContainerType_Vector_Vector_TcVnPoint2_DINT EXTENDS Node
VAR
    out : _GUID;
END_VAR

METHOD FB_init : BOOL
VAR_INPUT
	bInitRetains : BOOL; // if TRUE, the retain variables are initialized (warm start / cold start)
	bInCopyCode : BOOL;  // if TRUE, the instance afterwards gets moved into the copy code (online change)
END_VAR
AddOutput('out', out);
END_METHOD

METHOD PUBLIC  Clone : I_Node
VAR
	pNode : POINTER TO Node_ContainerType_Vector_Vector_TcVnPoint2_DINT;
END_VAR
pNode := __NEW(Node_ContainerType_Vector_Vector_TcVnPoint2_DINT);
Clone := pNode^;
END_METHOD

METHOD PROTECTED OnExecute
out.Value := ContainerType_Vector_Vector_TcVnPoint2_DINT;
END_METHOD

END_FUNCTION_BLOCK

// Nodes/Constants/Node_ContainerType_Vector_Vector_TcVnPoint2_REAL
{attribute 'linkalways'} 
{attribute 'no_explicit_call' := 'This FB is a CLASS and must be accessed using methods or properties'}
{attribute 'enable_dynamic_creation'}
FUNCTION_BLOCK Node_ContainerType_Vector_Vector_TcVnPoint2_REAL EXTENDS Node
VAR
    out : _GUID;
END_VAR

METHOD FB_init : BOOL
VAR_INPUT
	bInitRetains : BOOL; // if TRUE, the retain variables are initialized (warm start / cold start)
	bInCopyCode : BOOL;  // if TRUE, the instance afterwards gets moved into the copy code (online change)
END_VAR
AddOutput('out', out);
END_METHOD

METHOD PUBLIC  Clone : I_Node
VAR
	pNode : POINTER TO Node_ContainerType_Vector_Vector_TcVnPoint2_REAL;
END_VAR
pNode := __NEW(Node_ContainerType_Vector_Vector_TcVnPoint2_REAL);
Clone := pNode^;
END_METHOD

METHOD PROTECTED OnExecute
out.Value := ContainerType_Vector_Vector_TcVnPoint2_REAL;
END_METHOD

END_FUNCTION_BLOCK

// Nodes/Constants/Node_ContainerType_Vector_Vector_TcVnPoint3_REAL
{attribute 'linkalways'} 
{attribute 'no_explicit_call' := 'This FB is a CLASS and must be accessed using methods or properties'}
{attribute 'enable_dynamic_creation'}
FUNCTION_BLOCK Node_ContainerType_Vector_Vector_TcVnPoint3_REAL EXTENDS Node
VAR
    out : _GUID;
END_VAR

METHOD FB_init : BOOL
VAR_INPUT
	bInitRetains : BOOL; // if TRUE, the retain variables are initialized (warm start / cold start)
	bInCopyCode : BOOL;  // if TRUE, the instance afterwards gets moved into the copy code (online change)
END_VAR
AddOutput('out', out);
END_METHOD

METHOD PUBLIC  Clone : I_Node
VAR
	pNode : POINTER TO Node_ContainerType_Vector_Vector_TcVnPoint3_REAL;
END_VAR
pNode := __NEW(Node_ContainerType_Vector_Vector_TcVnPoint3_REAL);
Clone := pNode^;
END_METHOD

METHOD PROTECTED OnExecute
out.Value := ContainerType_Vector_Vector_TcVnPoint3_REAL;
END_METHOD

END_FUNCTION_BLOCK

// Nodes/Constants/Node_ContainerType_Vector_Vector_UDINT
{attribute 'linkalways'} 
{attribute 'no_explicit_call' := 'This FB is a CLASS and must be accessed using methods or properties'}
{attribute 'enable_dynamic_creation'}
FUNCTION_BLOCK Node_ContainerType_Vector_Vector_UDINT EXTENDS Node
VAR
    out : _GUID;
END_VAR

METHOD FB_init : BOOL
VAR_INPUT
	bInitRetains : BOOL; // if TRUE, the retain variables are initialized (warm start / cold start)
	bInCopyCode : BOOL;  // if TRUE, the instance afterwards gets moved into the copy code (online change)
END_VAR
AddOutput('out', out);
END_METHOD

METHOD PUBLIC  Clone : I_Node
VAR
	pNode : POINTER TO Node_ContainerType_Vector_Vector_UDINT;
END_VAR
pNode := __NEW(Node_ContainerType_Vector_Vector_UDINT);
Clone := pNode^;
END_METHOD

METHOD PROTECTED OnExecute
out.Value := ContainerType_Vector_Vector_UDINT;
END_METHOD

END_FUNCTION_BLOCK

// Nodes/Constants/Node_ContainerType_Vector_Vector_ULINT
{attribute 'linkalways'} 
{attribute 'no_explicit_call' := 'This FB is a CLASS and must be accessed using methods or properties'}
{attribute 'enable_dynamic_creation'}
FUNCTION_BLOCK Node_ContainerType_Vector_Vector_ULINT EXTENDS Node
VAR
    out : _GUID;
END_VAR

METHOD FB_init : BOOL
VAR_INPUT
	bInitRetains : BOOL; // if TRUE, the retain variables are initialized (warm start / cold start)
	bInCopyCode : BOOL;  // if TRUE, the instance afterwards gets moved into the copy code (online change)
END_VAR
AddOutput('out', out);
END_METHOD

METHOD PUBLIC  Clone : I_Node
VAR
	pNode : POINTER TO Node_ContainerType_Vector_Vector_ULINT;
END_VAR
pNode := __NEW(Node_ContainerType_Vector_Vector_ULINT);
Clone := pNode^;
END_METHOD

METHOD PROTECTED OnExecute
out.Value := ContainerType_Vector_Vector_ULINT;
END_METHOD

END_FUNCTION_BLOCK

// Nodes/Constants/Node_RGBA_BLACK
{attribute 'linkalways'} 
{attribute 'no_explicit_call' := 'This FB is a CLASS and must be accessed using methods or properties'}
{attribute 'enable_dynamic_creation'}
FUNCTION_BLOCK Node_RGBA_BLACK EXTENDS VisionNode
VAR
    out : _TcVnVector4_LREAL;
END_VAR

METHOD FB_init : BOOL
VAR_INPUT
	bInitRetains : BOOL; // if TRUE, the retain variables are initialized (warm start / cold start)
	bInCopyCode : BOOL;  // if TRUE, the instance afterwards gets moved into the copy code (online change)
END_VAR
AddOutput('out', out);
END_METHOD

METHOD PUBLIC  Clone : I_Node
VAR
	pNode : POINTER TO Node_RGBA_BLACK;
END_VAR
pNode := __NEW(Node_RGBA_BLACK);
Clone := pNode^;
END_METHOD

METHOD PROTECTED OnExecute
out.Value := GVL_COLOURS.RGBA_BLACK;
END_METHOD

METHOD PUBLIC PreExecutionCheck
VAR_INPUT
	Check : I_PreExecutionChecks;
END_VAR
END_METHOD

END_FUNCTION_BLOCK

// Nodes/Constants/Node_RGBA_BLUE
{attribute 'linkalways'} 
{attribute 'no_explicit_call' := 'This FB is a CLASS and must be accessed using methods or properties'}
{attribute 'enable_dynamic_creation'}
FUNCTION_BLOCK Node_RGBA_BLUE EXTENDS VisionNode
VAR
    out : _TcVnVector4_LREAL;
END_VAR

METHOD FB_init : BOOL
VAR_INPUT
	bInitRetains : BOOL; // if TRUE, the retain variables are initialized (warm start / cold start)
	bInCopyCode : BOOL;  // if TRUE, the instance afterwards gets moved into the copy code (online change)
END_VAR
AddOutput('out', out);
END_METHOD

METHOD PUBLIC  Clone : I_Node
VAR
	pNode : POINTER TO Node_RGBA_BLUE;
END_VAR
pNode := __NEW(Node_RGBA_BLUE);
Clone := pNode^;
END_METHOD

METHOD PROTECTED OnExecute
out.Value := GVL_COLOURS.RGBA_BLUE;
END_METHOD

METHOD PUBLIC PreExecutionCheck
VAR_INPUT
	Check : I_PreExecutionChecks;
END_VAR
END_METHOD

END_FUNCTION_BLOCK

// Nodes/Constants/Node_RGBA_CYAN
{attribute 'linkalways'} 
{attribute 'no_explicit_call' := 'This FB is a CLASS and must be accessed using methods or properties'}
{attribute 'enable_dynamic_creation'}
FUNCTION_BLOCK Node_RGBA_CYAN EXTENDS VisionNode
VAR
    out : _TcVnVector4_LREAL;
END_VAR

METHOD FB_init : BOOL
VAR_INPUT
	bInitRetains : BOOL; // if TRUE, the retain variables are initialized (warm start / cold start)
	bInCopyCode : BOOL;  // if TRUE, the instance afterwards gets moved into the copy code (online change)
END_VAR
AddOutput('out', out);
END_METHOD

METHOD PUBLIC  Clone : I_Node
VAR
	pNode : POINTER TO Node_RGBA_CYAN;
END_VAR
pNode := __NEW(Node_RGBA_CYAN);
Clone := pNode^;
END_METHOD

METHOD PROTECTED OnExecute
out.Value := GVL_COLOURS.RGBA_CYAN;
END_METHOD

METHOD PUBLIC PreExecutionCheck
VAR_INPUT
	Check : I_PreExecutionChecks;
END_VAR
END_METHOD

END_FUNCTION_BLOCK

// Nodes/Constants/Node_RGBA_GREEN
{attribute 'linkalways'} 
{attribute 'no_explicit_call' := 'This FB is a CLASS and must be accessed using methods or properties'}
{attribute 'enable_dynamic_creation'}
FUNCTION_BLOCK Node_RGBA_GREEN EXTENDS VisionNode
VAR
    out : _TcVnVector4_LREAL;
END_VAR

METHOD FB_init : BOOL
VAR_INPUT
	bInitRetains : BOOL; // if TRUE, the retain variables are initialized (warm start / cold start)
	bInCopyCode : BOOL;  // if TRUE, the instance afterwards gets moved into the copy code (online change)
END_VAR
AddOutput('out', out);
END_METHOD

METHOD PUBLIC  Clone : I_Node
VAR
	pNode : POINTER TO Node_RGBA_GREEN;
END_VAR
pNode := __NEW(Node_RGBA_GREEN);
Clone := pNode^;
END_METHOD

METHOD PROTECTED OnExecute
out.Value := GVL_COLOURS.RGBA_GREEN;
END_METHOD

METHOD PUBLIC PreExecutionCheck
VAR_INPUT
	Check : I_PreExecutionChecks;
END_VAR
END_METHOD

END_FUNCTION_BLOCK

// Nodes/Constants/Node_RGBA_MAGENTA
{attribute 'linkalways'} 
{attribute 'no_explicit_call' := 'This FB is a CLASS and must be accessed using methods or properties'}
{attribute 'enable_dynamic_creation'}
FUNCTION_BLOCK Node_RGBA_MAGENTA EXTENDS VisionNode
VAR
    out : _TcVnVector4_LREAL;
END_VAR

METHOD FB_init : BOOL
VAR_INPUT
	bInitRetains : BOOL; // if TRUE, the retain variables are initialized (warm start / cold start)
	bInCopyCode : BOOL;  // if TRUE, the instance afterwards gets moved into the copy code (online change)
END_VAR
AddOutput('out', out);
END_METHOD

METHOD PUBLIC  Clone : I_Node
VAR
	pNode : POINTER TO Node_RGBA_MAGENTA;
END_VAR
pNode := __NEW(Node_RGBA_MAGENTA);
Clone := pNode^;
END_METHOD

METHOD PROTECTED OnExecute
out.Value := GVL_COLOURS.RGBA_MAGENTA;
END_METHOD

METHOD PUBLIC PreExecutionCheck
VAR_INPUT
	Check : I_PreExecutionChecks;
END_VAR
END_METHOD

END_FUNCTION_BLOCK

// Nodes/Constants/Node_RGBA_RANDOM
{attribute 'linkalways'} 
{attribute 'no_explicit_call' := 'This FB is a CLASS and must be accessed using methods or properties'}
{attribute 'enable_dynamic_creation'}
FUNCTION_BLOCK Node_RGBA_RANDOM EXTENDS VisionNode
VAR
    out : _TcVnVector4_LREAL;
END_VAR

METHOD FB_init : BOOL
VAR_INPUT
	bInitRetains : BOOL; // if TRUE, the retain variables are initialized (warm start / cold start)
	bInCopyCode : BOOL;  // if TRUE, the instance afterwards gets moved into the copy code (online change)
END_VAR
AddOutput('out', out);
END_METHOD

METHOD PUBLIC  Clone : I_Node
VAR
	pNode : POINTER TO Node_RGBA_RANDOM;
END_VAR
pNode := __NEW(Node_RGBA_RANDOM);
Clone := pNode^;
END_METHOD

METHOD PROTECTED OnExecute
out.Value := GVL_COLOURS.RGBA_RANDOM;
END_METHOD

METHOD PUBLIC PreExecutionCheck
VAR_INPUT
	Check : I_PreExecutionChecks;
END_VAR
END_METHOD

END_FUNCTION_BLOCK

// Nodes/Constants/Node_RGBA_RED
{attribute 'linkalways'} 
{attribute 'no_explicit_call' := 'This FB is a CLASS and must be accessed using methods or properties'}
{attribute 'enable_dynamic_creation'}
FUNCTION_BLOCK Node_RGBA_RED EXTENDS VisionNode
VAR
    out : _TcVnVector4_LREAL;
END_VAR

METHOD FB_init : BOOL
VAR_INPUT
	bInitRetains : BOOL; // if TRUE, the retain variables are initialized (warm start / cold start)
	bInCopyCode : BOOL;  // if TRUE, the instance afterwards gets moved into the copy code (online change)
END_VAR
AddOutput('out', out);
END_METHOD

METHOD PUBLIC  Clone : I_Node
VAR
	pNode : POINTER TO Node_RGBA_RED;
END_VAR
pNode := __NEW(Node_RGBA_RED);
Clone := pNode^;
END_METHOD

METHOD PROTECTED OnExecute
out.Value := GVL_COLOURS.RGBA_RED;
END_METHOD

METHOD PUBLIC PreExecutionCheck
VAR_INPUT
	Check : I_PreExecutionChecks;
END_VAR
END_METHOD

END_FUNCTION_BLOCK

// Nodes/Constants/Node_RGBA_WHITE
{attribute 'linkalways'} 
{attribute 'no_explicit_call' := 'This FB is a CLASS and must be accessed using methods or properties'}
{attribute 'enable_dynamic_creation'}
FUNCTION_BLOCK Node_RGBA_WHITE EXTENDS VisionNode
VAR
    out : _TcVnVector4_LREAL;
END_VAR

METHOD FB_init : BOOL
VAR_INPUT
	bInitRetains : BOOL; // if TRUE, the retain variables are initialized (warm start / cold start)
	bInCopyCode : BOOL;  // if TRUE, the instance afterwards gets moved into the copy code (online change)
END_VAR
AddOutput('out', out);
END_METHOD

METHOD PUBLIC  Clone : I_Node
VAR
	pNode : POINTER TO Node_RGBA_WHITE;
END_VAR
pNode := __NEW(Node_RGBA_WHITE);
Clone := pNode^;
END_METHOD

METHOD PROTECTED OnExecute
out.Value := GVL_COLOURS.RGBA_WHITE;
END_METHOD

METHOD PUBLIC PreExecutionCheck
VAR_INPUT
	Check : I_PreExecutionChecks;
END_VAR
END_METHOD

END_FUNCTION_BLOCK

// Nodes/Constants/Node_RGBA_YELLOW
{attribute 'linkalways'} 
{attribute 'no_explicit_call' := 'This FB is a CLASS and must be accessed using methods or properties'}
{attribute 'enable_dynamic_creation'}
FUNCTION_BLOCK Node_RGBA_YELLOW EXTENDS VisionNode
VAR
    out : _TcVnVector4_LREAL;
END_VAR

METHOD FB_init : BOOL
VAR_INPUT
	bInitRetains : BOOL; // if TRUE, the retain variables are initialized (warm start / cold start)
	bInCopyCode : BOOL;  // if TRUE, the instance afterwards gets moved into the copy code (online change)
END_VAR
AddOutput('out', out);
END_METHOD

METHOD PUBLIC  Clone : I_Node
VAR
	pNode : POINTER TO Node_RGBA_YELLOW;
END_VAR
pNode := __NEW(Node_RGBA_YELLOW);
Clone := pNode^;
END_METHOD

METHOD PROTECTED OnExecute
out.Value := GVL_COLOURS.RGBA_YELLOW;
END_METHOD

METHOD PUBLIC PreExecutionCheck
VAR_INPUT
	Check : I_PreExecutionChecks;
END_VAR
END_METHOD

END_FUNCTION_BLOCK

// Nodes/Container Statistics/MaxElementwise/Node_F_VN_MaxElementElementwise_DINT
{attribute 'linkalways'} 
{attribute 'no_explicit_call' := 'This FB is a CLASS and must be accessed using methods or properties'}
{attribute 'enable_dynamic_creation'}
FUNCTION_BLOCK Node_F_VN_MaxElementElementwise_DINT EXTENDS VisionNode
VAR
    ipContainer : _ITcVnContainer;
    nMax : _DINT(0);
    hrPrev : _HRESULT(S_OK);
    hresult : _HRESULT(S_OK);
END_VAR

METHOD FB_init : BOOL
VAR_INPUT
	bInitRetains : BOOL; // if TRUE, the retain variables are initialized (warm start / cold start)
	bInCopyCode : BOOL;  // if TRUE, the instance afterwards gets moved into the copy code (online change)
END_VAR
AddInput('ipContainer', ipContainer);
AddInput('hrPrev', hrPrev);
AddOutput('ipContainer', ipContainer);
AddOutput('nMax', nMax);
AddOutput('hresult',hresult);
END_METHOD

METHOD PUBLIC  Clone : I_Node
VAR
	pNode : POINTER TO Node_F_VN_MaxElementElementwise_DINT;
END_VAR
pNode := __NEW(Node_F_VN_MaxElementElementwise_DINT);
Clone := pNode^;
END_METHOD

METHOD PROTECTED OnExecute
hresult.Value := F_VN_MaxElementElementwise_DINT(
    ipContainer := ipContainer.Value,
    nMax := nMax.Value,
    hrPrev:= hrPrev.Value);
END_METHOD

METHOD PUBLIC PreExecutionCheck
VAR_INPUT
	Check : I_PreExecutionChecks;
END_VAR
VAR
    name : STRING;
END_VAR
Check.IsTrue(ipContainer.IsValid, 'ipContainer must be a valid container');
Check.IsTrue(ipContainer.IsType(TC_GLOBAL_CONST_LIST.ContainerType_Vector_DINT), 'ipContainer contains incorrect type');
END_METHOD

END_FUNCTION_BLOCK

// Nodes/Container Statistics/MaxElementwise/Node_F_VN_MaxElementElementwise_INT
{attribute 'linkalways'} 
{attribute 'no_explicit_call' := 'This FB is a CLASS and must be accessed using methods or properties'}
{attribute 'enable_dynamic_creation'}
FUNCTION_BLOCK Node_F_VN_MaxElementElementwise_INT EXTENDS VisionNode
VAR
    ipContainer : _ITcVnContainer;
    nMax : _INT(0);
    hrPrev : _HRESULT(S_OK);
    hresult : _HRESULT(S_OK);
END_VAR

METHOD FB_init : BOOL
VAR_INPUT
	bInitRetains : BOOL; // if TRUE, the retain variables are initialized (warm start / cold start)
	bInCopyCode : BOOL;  // if TRUE, the instance afterwards gets moved into the copy code (online change)
END_VAR
AddInput('ipContainer', ipContainer);
AddInput('hrPrev', hrPrev);
AddOutput('ipContainer', ipContainer);
AddOutput('nMax', nMax);
AddOutput('hresult',hresult);
END_METHOD

METHOD PUBLIC  Clone : I_Node
VAR
	pNode : POINTER TO Node_F_VN_MaxElementElementwise_INT;
END_VAR
pNode := __NEW(Node_F_VN_MaxElementElementwise_INT);
Clone := pNode^;
END_METHOD

METHOD PROTECTED OnExecute
hresult.Value := F_VN_MaxElementElementwise_INT(
    ipContainer := ipContainer.Value,
    nMax := nMax.Value,
    hrPrev:= hrPrev.Value);
END_METHOD

METHOD PUBLIC PreExecutionCheck
VAR_INPUT
	Check : I_PreExecutionChecks;
END_VAR
Check.IsTrue(ipContainer.IsValid, 'ipContainer must be a valid container');
Check.IsTrue(ipContainer.IsType(TC_GLOBAL_CONST_LIST.ContainerType_Vector_INT), 'ipContainer contains incorrect type');
END_METHOD

END_FUNCTION_BLOCK

// Nodes/Container Statistics/MaxElementwise/Node_F_VN_MaxElementElementwise_LREAL
{attribute 'linkalways'} 
{attribute 'no_explicit_call' := 'This FB is a CLASS and must be accessed using methods or properties'}
{attribute 'enable_dynamic_creation'}
FUNCTION_BLOCK Node_F_VN_MaxElementElementwise_LREAL EXTENDS VisionNode
VAR
    ipContainer : _ITcVnContainer;
    fMax : _LREAL(0.0);
    hrPrev : _HRESULT(S_OK);
    hresult : _HRESULT(S_OK);
END_VAR

METHOD FB_init : BOOL
VAR_INPUT
	bInitRetains : BOOL; // if TRUE, the retain variables are initialized (warm start / cold start)
	bInCopyCode : BOOL;  // if TRUE, the instance afterwards gets moved into the copy code (online change)
END_VAR
AddInput('ipContainer', ipContainer);
AddInput('hrPrev', hrPrev);
AddOutput('ipContainer', ipContainer);
AddOutput('fMax', fMax);
AddOutput('hresult',hresult);
END_METHOD

METHOD PUBLIC  Clone : I_Node
VAR
	pNode : POINTER TO Node_F_VN_MaxElementElementwise_LREAL;
END_VAR
pNode := __NEW(Node_F_VN_MaxElementElementwise_LREAL);
Clone := pNode^;
END_METHOD

METHOD PROTECTED OnExecute
hresult.Value := F_VN_MaxElementElementwise_LREAL(
    ipContainer := ipContainer.Value,
    fMax := fMax.Value,
    hrPrev:= hrPrev.Value);
END_METHOD

METHOD PUBLIC PreExecutionCheck
VAR_INPUT
	Check : I_PreExecutionChecks;
END_VAR
Check.IsTrue(ipContainer.IsValid, 'ipContainer must be a valid container');
Check.IsTrue(ipContainer.IsType(TC_GLOBAL_CONST_LIST.ContainerType_Vector_LREAL), 'ipContainer contains incorrect type');
END_METHOD

END_FUNCTION_BLOCK

// Nodes/Container Statistics/MaxElementwise/Node_F_VN_MaxElementElementwise_REAL
{attribute 'linkalways'} 
{attribute 'no_explicit_call' := 'This FB is a CLASS and must be accessed using methods or properties'}
{attribute 'enable_dynamic_creation'}
FUNCTION_BLOCK Node_F_VN_MaxElementElementwise_REAL EXTENDS VisionNode
VAR
    ipContainer : _ITcVnContainer;
    fMax : _REAL(0.0);
    hrPrev : _HRESULT(S_OK);
    hresult : _HRESULT(S_OK);
END_VAR

METHOD FB_init : BOOL
VAR_INPUT
	bInitRetains : BOOL; // if TRUE, the retain variables are initialized (warm start / cold start)
	bInCopyCode : BOOL;  // if TRUE, the instance afterwards gets moved into the copy code (online change)
END_VAR
AddInput('ipContainer', ipContainer);
AddInput('hrPrev', hrPrev);
AddOutput('ipContainer', ipContainer);
AddOutput('fMax', fMax);
AddOutput('hresult',hresult);
END_METHOD

METHOD PUBLIC  Clone : I_Node
VAR
	pNode : POINTER TO Node_F_VN_MaxElementElementwise_REAL;
END_VAR
pNode := __NEW(Node_F_VN_MaxElementElementwise_REAL);
Clone := pNode^;
END_METHOD

METHOD PROTECTED OnExecute
hresult.Value := F_VN_MaxElementElementwise_REAL(
    ipContainer := ipContainer.Value,
    fMax := fMax.Value,
    hrPrev:= hrPrev.Value);
END_METHOD

METHOD PUBLIC PreExecutionCheck
VAR_INPUT
	Check : I_PreExecutionChecks;
END_VAR
Check.IsTrue(ipContainer.IsValid, 'ipContainer must be a valid container');
Check.IsTrue(ipContainer.IsType(TC_GLOBAL_CONST_LIST.ContainerType_Vector_REAL), 'ipContainer contains incorrect type');
END_METHOD

END_FUNCTION_BLOCK

// Nodes/Container Statistics/MaxElementwise/Node_F_VN_MaxElementElementwise_SINT
{attribute 'linkalways'} 
{attribute 'no_explicit_call' := 'This FB is a CLASS and must be accessed using methods or properties'}
{attribute 'enable_dynamic_creation'}
FUNCTION_BLOCK Node_F_VN_MaxElementElementwise_SINT EXTENDS VisionNode
VAR
    ipContainer : _ITcVnContainer;
    nMax : _SINT(0);
    hrPrev : _HRESULT(S_OK);
    hresult : _HRESULT(S_OK);
END_VAR

METHOD FB_init : BOOL
VAR_INPUT
	bInitRetains : BOOL; // if TRUE, the retain variables are initialized (warm start / cold start)
	bInCopyCode : BOOL;  // if TRUE, the instance afterwards gets moved into the copy code (online change)
END_VAR
AddInput('ipContainer', ipContainer);
AddInput('hrPrev', hrPrev);
AddOutput('ipContainer', ipContainer);
AddOutput('nMax', nMax);
AddOutput('hresult',hresult);
END_METHOD

METHOD PUBLIC  Clone : I_Node
VAR
	pNode : POINTER TO Node_F_VN_MaxElementElementwise_SINT;
END_VAR
pNode := __NEW(Node_F_VN_MaxElementElementwise_SINT);
Clone := pNode^;
END_METHOD

METHOD PROTECTED OnExecute
hresult.Value := F_VN_MaxElementElementwise_SINT(
    ipContainer := ipContainer.Value,
    nMax := nMax.Value,
    hrPrev:= hrPrev.Value);
END_METHOD

METHOD PUBLIC PreExecutionCheck
VAR_INPUT
	Check : I_PreExecutionChecks;
END_VAR
Check.IsTrue(ipContainer.IsValid, 'ipContainer must be a valid container');
Check.IsTrue(ipContainer.IsType(TC_GLOBAL_CONST_LIST.ContainerType_Vector_SINT), 'ipContainer contains incorrect type');
END_METHOD

END_FUNCTION_BLOCK

// Nodes/Container Statistics/MaxElementwise/Node_F_VN_MaxElementElementwise_TcVnPoint2_DINT
{attribute 'linkalways'} 
{attribute 'no_explicit_call' := 'This FB is a CLASS and must be accessed using methods or properties'}
{attribute 'enable_dynamic_creation'}
FUNCTION_BLOCK Node_F_VN_MaxElementElementwise_TcVnPoint2_DINT EXTENDS VisionNode
VAR
    ipContainer : _ITcVnContainer;
    aMax : _TcVnPoint2_DINT;
    hrPrev : _HRESULT(S_OK);
    hresult : _HRESULT(S_OK);
END_VAR

METHOD FB_init : BOOL
VAR_INPUT
	bInitRetains : BOOL; // if TRUE, the retain variables are initialized (warm start / cold start)
	bInCopyCode : BOOL;  // if TRUE, the instance afterwards gets moved into the copy code (online change)
END_VAR
AddInput('ipContainer', ipContainer);
AddInput('hrPrev', hrPrev);
AddOutput('ipContainer', ipContainer);
AddOutput('aMax', aMax);
AddOutput('hresult',hresult);
END_METHOD

METHOD PUBLIC  Clone : I_Node
VAR
	pNode : POINTER TO Node_F_VN_MaxElementElementwise_TcVnPoint2_DINT;
END_VAR
pNode := __NEW(Node_F_VN_MaxElementElementwise_TcVnPoint2_DINT);
Clone := pNode^;
END_METHOD

METHOD PROTECTED OnExecute
hresult.Value := F_VN_MaxElementElementwise_TcVnPoint2_DINT(
    ipContainer := ipContainer.Value,
    aMax := aMax.Value,
    hrPrev:= hrPrev.Value);
END_METHOD

METHOD PUBLIC PreExecutionCheck
VAR_INPUT
	Check : I_PreExecutionChecks;
END_VAR
Check.IsTrue(ipContainer.IsValid, 'ipContainer must be a valid container');
Check.IsTrue(ipContainer.IsType(TC_GLOBAL_CONST_LIST.ContainerType_Vector_TcVnPoint2_DINT), 'ipContainer contains incorrect type');
END_METHOD

END_FUNCTION_BLOCK

// Nodes/Container Statistics/MaxElementwise/Node_F_VN_MaxElementElementwise_TcVnPoint2_LREAL
{attribute 'linkalways'} 
{attribute 'no_explicit_call' := 'This FB is a CLASS and must be accessed using methods or properties'}
{attribute 'enable_dynamic_creation'}
FUNCTION_BLOCK Node_F_VN_MaxElementElementwise_TcVnPoint2_LREAL EXTENDS VisionNode
VAR
    ipContainer : _ITcVnContainer;
    aMax : _TcVnPoint2_LREAL;
    hrPrev : _HRESULT(S_OK);
    hresult : _HRESULT(S_OK);
END_VAR

METHOD FB_init : BOOL
VAR_INPUT
	bInitRetains : BOOL; // if TRUE, the retain variables are initialized (warm start / cold start)
	bInCopyCode : BOOL;  // if TRUE, the instance afterwards gets moved into the copy code (online change)
END_VAR
AddInput('ipContainer', ipContainer);
AddInput('hrPrev', hrPrev);
AddOutput('ipContainer', ipContainer);
AddOutput('aMax', aMax);
AddOutput('hresult',hresult);
END_METHOD

METHOD PUBLIC  Clone : I_Node
VAR
	pNode : POINTER TO Node_F_VN_MaxElementElementwise_TcVnPoint2_LREAL;
END_VAR
pNode := __NEW(Node_F_VN_MaxElementElementwise_TcVnPoint2_LREAL);
Clone := pNode^;
END_METHOD

METHOD PROTECTED OnExecute
hresult.Value := F_VN_MaxElementElementwise_TcVnPoint2_LREAL(
    ipContainer := ipContainer.Value,
    aMax := aMax.Value,
    hrPrev:= hrPrev.Value);
END_METHOD

METHOD PUBLIC PreExecutionCheck
VAR_INPUT
	Check : I_PreExecutionChecks;
END_VAR
Check.IsTrue(ipContainer.IsValid, 'ipContainer must be a valid container');
Check.IsTrue(ipContainer.IsType(TC_GLOBAL_CONST_LIST.ContainerType_Vector_TcVnPoint2_LREAL), 'ipContainer contains incorrect type');
END_METHOD

END_FUNCTION_BLOCK

// Nodes/Container Statistics/MaxElementwise/Node_F_VN_MaxElementElementwise_TcVnPoint2_REAL
{attribute 'linkalways'} 
{attribute 'no_explicit_call' := 'This FB is a CLASS and must be accessed using methods or properties'}
{attribute 'enable_dynamic_creation'}
FUNCTION_BLOCK Node_F_VN_MaxElementElementwise_TcVnPoint2_REAL EXTENDS VisionNode
VAR
    ipContainer : _ITcVnContainer;
    aMax : _TcVnPoint2_REAL;
    hrPrev : _HRESULT(S_OK);
    hresult : _HRESULT(S_OK);
END_VAR

METHOD FB_init : BOOL
VAR_INPUT
	bInitRetains : BOOL; // if TRUE, the retain variables are initialized (warm start / cold start)
	bInCopyCode : BOOL;  // if TRUE, the instance afterwards gets moved into the copy code (online change)
END_VAR
AddInput('ipContainer', ipContainer);
AddInput('hrPrev', hrPrev);
AddOutput('ipContainer', ipContainer);
AddOutput('aMax', aMax);
AddOutput('hresult',hresult);
END_METHOD

METHOD PUBLIC  Clone : I_Node
VAR
	pNode : POINTER TO Node_F_VN_MaxElementElementwise_TcVnPoint2_REAL;
END_VAR
pNode := __NEW(Node_F_VN_MaxElementElementwise_TcVnPoint2_REAL);
Clone := pNode^;
END_METHOD

METHOD PROTECTED OnExecute
hresult.Value := F_VN_MaxElementElementwise_TcVnPoint2_REAL(
    ipContainer := ipContainer.Value,
    aMax := aMax.Value,
    hrPrev:= hrPrev.Value);
END_METHOD

METHOD PUBLIC PreExecutionCheck
VAR_INPUT
	Check : I_PreExecutionChecks;
END_VAR
Check.IsTrue(ipContainer.IsValid, 'ipContainer must be a valid container');
Check.IsTrue(ipContainer.IsType(TC_GLOBAL_CONST_LIST.ContainerType_Vector_TcVnPoint2_REAL), 'ipContainer contains incorrect type');
END_METHOD

END_FUNCTION_BLOCK

// Nodes/Container Statistics/MaxElementwise/Node_F_VN_MaxElementElementwise_TcVnPoint3_LREAL
{attribute 'linkalways'} 
{attribute 'no_explicit_call' := 'This FB is a CLASS and must be accessed using methods or properties'}
{attribute 'enable_dynamic_creation'}
FUNCTION_BLOCK Node_F_VN_MaxElementElementwise_TcVnPoint3_LREAL EXTENDS VisionNode
VAR
    ipContainer : _ITcVnContainer;
    aMax : _TcVnPoint3_LREAL;
    hrPrev : _HRESULT(S_OK);
    hresult : _HRESULT(S_OK);
END_VAR

METHOD FB_init : BOOL
VAR_INPUT
	bInitRetains : BOOL; // if TRUE, the retain variables are initialized (warm start / cold start)
	bInCopyCode : BOOL;  // if TRUE, the instance afterwards gets moved into the copy code (online change)
END_VAR
AddInput('ipContainer', ipContainer);
AddInput('hrPrev', hrPrev);
AddOutput('ipContainer', ipContainer);
AddOutput('aMax', aMax);
AddOutput('hresult',hresult);
END_METHOD

METHOD PUBLIC  Clone : I_Node
VAR
	pNode : POINTER TO Node_F_VN_MaxElementElementwise_TcVnPoint3_LREAL;
END_VAR
pNode := __NEW(Node_F_VN_MaxElementElementwise_TcVnPoint3_LREAL);
Clone := pNode^;
END_METHOD

METHOD PROTECTED OnExecute
hresult.Value := F_VN_MaxElementElementwise_TcVnPoint3_LREAL(
    ipContainer := ipContainer.Value,
    aMax := aMax.Value,
    hrPrev:= hrPrev.Value);
END_METHOD

METHOD PUBLIC PreExecutionCheck
VAR_INPUT
	Check : I_PreExecutionChecks;
END_VAR
Check.IsTrue(ipContainer.IsValid, 'ipContainer must be a valid container');
Check.IsTrue(ipContainer.IsType(TC_GLOBAL_CONST_LIST.ContainerType_Vector_TcVnPoint3_LREAL), 'ipContainer contains incorrect type');
END_METHOD

END_FUNCTION_BLOCK

// Nodes/Container Statistics/MaxElementwise/Node_F_VN_MaxElementElementwise_TcVnPoint3_REAL
{attribute 'linkalways'} 
{attribute 'no_explicit_call' := 'This FB is a CLASS and must be accessed using methods or properties'}
{attribute 'enable_dynamic_creation'}
FUNCTION_BLOCK Node_F_VN_MaxElementElementwise_TcVnPoint3_REAL EXTENDS VisionNode
VAR
    ipContainer : _ITcVnContainer;
    aMax : _TcVnPoint3_REAL;
    hrPrev : _HRESULT(S_OK);
    hresult : _HRESULT(S_OK);
END_VAR

METHOD FB_init : BOOL
VAR_INPUT
	bInitRetains : BOOL; // if TRUE, the retain variables are initialized (warm start / cold start)
	bInCopyCode : BOOL;  // if TRUE, the instance afterwards gets moved into the copy code (online change)
END_VAR
AddInput('ipContainer', ipContainer);
AddInput('hrPrev', hrPrev);
AddOutput('ipContainer', ipContainer);
AddOutput('aMax', aMax);
AddOutput('hresult',hresult);
END_METHOD

METHOD PUBLIC  Clone : I_Node
VAR
	pNode : POINTER TO Node_F_VN_MaxElementElementwise_TcVnPoint3_REAL;
END_VAR
pNode := __NEW(Node_F_VN_MaxElementElementwise_TcVnPoint3_REAL);
Clone := pNode^;
END_METHOD

METHOD PROTECTED OnExecute
hresult.Value := F_VN_MaxElementElementwise_TcVnPoint3_REAL(
    ipContainer := ipContainer.Value,
    aMax := aMax.Value,
    hrPrev:= hrPrev.Value);
END_METHOD

METHOD PUBLIC PreExecutionCheck
VAR_INPUT
	Check : I_PreExecutionChecks;
END_VAR
Check.IsTrue(ipContainer.IsValid, 'ipContainer must be a valid container');
Check.IsTrue(ipContainer.IsType(TC_GLOBAL_CONST_LIST.ContainerType_Vector_TcVnPoint3_REAL), 'ipContainer contains incorrect type');
END_METHOD

END_FUNCTION_BLOCK

// Nodes/Container Statistics/MaxElementwise/Node_F_VN_MaxElementElementwise_TcVnVector2_DINT
{attribute 'linkalways'} 
{attribute 'no_explicit_call' := 'This FB is a CLASS and must be accessed using methods or properties'}
{attribute 'enable_dynamic_creation'}
FUNCTION_BLOCK Node_F_VN_MaxElementElementwise_TcVnVector2_DINT EXTENDS VisionNode
VAR
    ipContainer : _ITcVnContainer;
    aMax : _TcVnVector2_DINT;
    hrPrev : _HRESULT(S_OK);
    hresult : _HRESULT(S_OK);
END_VAR

METHOD FB_init : BOOL
VAR_INPUT
	bInitRetains : BOOL; // if TRUE, the retain variables are initialized (warm start / cold start)
	bInCopyCode : BOOL;  // if TRUE, the instance afterwards gets moved into the copy code (online change)
END_VAR
AddInput('ipContainer', ipContainer);
AddInput('hrPrev', hrPrev);
AddOutput('ipContainer', ipContainer);
AddOutput('aMax', aMax);
AddOutput('hresult',hresult);
END_METHOD

METHOD PUBLIC  Clone : I_Node
VAR
	pNode : POINTER TO Node_F_VN_MaxElementElementwise_TcVnVector2_DINT;
END_VAR
pNode := __NEW(Node_F_VN_MaxElementElementwise_TcVnVector2_DINT);
Clone := pNode^;
END_METHOD

METHOD PROTECTED OnExecute
hresult.Value := F_VN_MaxElementElementwise_TcVnVector2_DINT(
    ipContainer := ipContainer.Value,
    aMax := aMax.Value,
    hrPrev:= hrPrev.Value);
END_METHOD

METHOD PUBLIC PreExecutionCheck
VAR_INPUT
	Check : I_PreExecutionChecks;
END_VAR
Check.IsTrue(ipContainer.IsValid, 'ipContainer must be a valid container');
Check.IsTrue(ipContainer.IsType(TC_GLOBAL_CONST_LIST.ContainerType_Vector_TcVnVector2_DINT), 'ipContainer contains incorrect type');
END_METHOD

END_FUNCTION_BLOCK

// Nodes/Container Statistics/MaxElementwise/Node_F_VN_MaxElementElementwise_TcVnVector2_INT
{attribute 'linkalways'} 
{attribute 'no_explicit_call' := 'This FB is a CLASS and must be accessed using methods or properties'}
{attribute 'enable_dynamic_creation'}
FUNCTION_BLOCK Node_F_VN_MaxElementElementwise_TcVnVector2_INT EXTENDS VisionNode
VAR
    ipContainer : _ITcVnContainer;
    aMax : _TcVnVector2_INT;
    hrPrev : _HRESULT(S_OK);
    hresult : _HRESULT(S_OK);
END_VAR

METHOD FB_init : BOOL
VAR_INPUT
	bInitRetains : BOOL; // if TRUE, the retain variables are initialized (warm start / cold start)
	bInCopyCode : BOOL;  // if TRUE, the instance afterwards gets moved into the copy code (online change)
END_VAR
AddInput('ipContainer', ipContainer);
AddInput('hrPrev', hrPrev);
AddOutput('ipContainer', ipContainer);
AddOutput('aMax', aMax);
AddOutput('hresult',hresult);
END_METHOD

METHOD PUBLIC  Clone : I_Node
VAR
	pNode : POINTER TO Node_F_VN_MaxElementElementwise_TcVnVector2_INT;
END_VAR
pNode := __NEW(Node_F_VN_MaxElementElementwise_TcVnVector2_INT);
Clone := pNode^;
END_METHOD

METHOD PROTECTED OnExecute
hresult.Value := F_VN_MaxElementElementwise_TcVnVector2_INT(
    ipContainer := ipContainer.Value,
    aMax := aMax.Value,
    hrPrev:= hrPrev.Value);
END_METHOD

METHOD PUBLIC PreExecutionCheck
VAR_INPUT
	Check : I_PreExecutionChecks;
END_VAR
Check.IsTrue(ipContainer.IsValid, 'ipContainer must be a valid container');
Check.IsTrue(ipContainer.IsType(TC_GLOBAL_CONST_LIST.ContainerType_Vector_TcVnVector2_INT), 'ipContainer contains incorrect type');
END_METHOD

END_FUNCTION_BLOCK

// Nodes/Container Statistics/MaxElementwise/Node_F_VN_MaxElementElementwise_TcVnVector2_REAL
{attribute 'linkalways'} 
{attribute 'no_explicit_call' := 'This FB is a CLASS and must be accessed using methods or properties'}
{attribute 'enable_dynamic_creation'}
FUNCTION_BLOCK Node_F_VN_MaxElementElementwise_TcVnVector2_REAL EXTENDS VisionNode
VAR
    ipContainer : _ITcVnContainer;
    aMax : _TcVnVector2_REAL;
    hrPrev : _HRESULT(S_OK);
    hresult : _HRESULT(S_OK);
END_VAR

METHOD FB_init : BOOL
VAR_INPUT
	bInitRetains : BOOL; // if TRUE, the retain variables are initialized (warm start / cold start)
	bInCopyCode : BOOL;  // if TRUE, the instance afterwards gets moved into the copy code (online change)
END_VAR
AddInput('ipContainer', ipContainer);
AddInput('hrPrev', hrPrev);
AddOutput('ipContainer', ipContainer);
AddOutput('aMax', aMax);
AddOutput('hresult',hresult);
END_METHOD

METHOD PUBLIC  Clone : I_Node
VAR
	pNode : POINTER TO Node_F_VN_MaxElementElementwise_TcVnVector2_REAL;
END_VAR
pNode := __NEW(Node_F_VN_MaxElementElementwise_TcVnVector2_REAL);
Clone := pNode^;
END_METHOD

METHOD PROTECTED OnExecute
hresult.Value := F_VN_MaxElementElementwise_TcVnVector2_REAL(
    ipContainer := ipContainer.Value,
    aMax := aMax.Value,
    hrPrev:= hrPrev.Value);
END_METHOD

METHOD PUBLIC PreExecutionCheck
VAR_INPUT
	Check : I_PreExecutionChecks;
END_VAR
Check.IsTrue(ipContainer.IsValid, 'ipContainer must be a valid container');
Check.IsTrue(ipContainer.IsType(TC_GLOBAL_CONST_LIST.ContainerType_Vector_TcVnVector2_REAL), 'ipContainer contains incorrect type');
END_METHOD

END_FUNCTION_BLOCK

// Nodes/Container Statistics/MaxElementwise/Node_F_VN_MaxElementElementwise_TcVnVector2_SINT
{attribute 'linkalways'} 
{attribute 'no_explicit_call' := 'This FB is a CLASS and must be accessed using methods or properties'}
{attribute 'enable_dynamic_creation'}
FUNCTION_BLOCK Node_F_VN_MaxElementElementwise_TcVnVector2_SINT EXTENDS VisionNode
VAR
    ipContainer : _ITcVnContainer;
    aMax : _TcVnVector2_SINT;
    hrPrev : _HRESULT(S_OK);
    hresult : _HRESULT(S_OK);
END_VAR

METHOD FB_init : BOOL
VAR_INPUT
	bInitRetains : BOOL; // if TRUE, the retain variables are initialized (warm start / cold start)
	bInCopyCode : BOOL;  // if TRUE, the instance afterwards gets moved into the copy code (online change)
END_VAR
AddInput('ipContainer', ipContainer);
AddInput('hrPrev', hrPrev);
AddOutput('ipContainer', ipContainer);
AddOutput('aMax', aMax);
AddOutput('hresult',hresult);
END_METHOD

METHOD PUBLIC  Clone : I_Node
VAR
	pNode : POINTER TO Node_F_VN_MaxElementElementwise_TcVnVector2_SINT;
END_VAR
pNode := __NEW(Node_F_VN_MaxElementElementwise_TcVnVector2_SINT);
Clone := pNode^;
END_METHOD

METHOD PROTECTED OnExecute
hresult.Value := F_VN_MaxElementElementwise_TcVnVector2_SINT(
    ipContainer := ipContainer.Value,
    aMax := aMax.Value,
    hrPrev:= hrPrev.Value);
END_METHOD

METHOD PUBLIC PreExecutionCheck
VAR_INPUT
	Check : I_PreExecutionChecks;
END_VAR
Check.IsTrue(ipContainer.IsValid, 'ipContainer must be a valid container');
Check.IsTrue(ipContainer.IsType(TC_GLOBAL_CONST_LIST.ContainerType_Vector_TcVnVector2_SINT), 'ipContainer contains incorrect type');
END_METHOD

END_FUNCTION_BLOCK

// Nodes/Container Statistics/MaxElementwise/Node_F_VN_MaxElementElementwise_TcVnVector2_UINT
{attribute 'linkalways'} 
{attribute 'no_explicit_call' := 'This FB is a CLASS and must be accessed using methods or properties'}
{attribute 'enable_dynamic_creation'}
FUNCTION_BLOCK Node_F_VN_MaxElementElementwise_TcVnVector2_UINT EXTENDS VisionNode
VAR
    ipContainer : _ITcVnContainer;
    aMax : _TcVnVector2_UINT;
    hrPrev : _HRESULT(S_OK);
    hresult : _HRESULT(S_OK);
END_VAR

METHOD FB_init : BOOL
VAR_INPUT
	bInitRetains : BOOL; // if TRUE, the retain variables are initialized (warm start / cold start)
	bInCopyCode : BOOL;  // if TRUE, the instance afterwards gets moved into the copy code (online change)
END_VAR
AddInput('ipContainer', ipContainer);
AddInput('hrPrev', hrPrev);
AddOutput('ipContainer', ipContainer);
AddOutput('aMax', aMax);
AddOutput('hresult',hresult);
END_METHOD

METHOD PUBLIC  Clone : I_Node
VAR
	pNode : POINTER TO Node_F_VN_MaxElementElementwise_TcVnVector2_UINT;
END_VAR
pNode := __NEW(Node_F_VN_MaxElementElementwise_TcVnVector2_UINT);
Clone := pNode^;
END_METHOD

METHOD PROTECTED OnExecute
hresult.Value := F_VN_MaxElementElementwise_TcVnVector2_UINT(
    ipContainer := ipContainer.Value,
    aMax := aMax.Value,
    hrPrev:= hrPrev.Value);
END_METHOD

METHOD PUBLIC PreExecutionCheck
VAR_INPUT
	Check : I_PreExecutionChecks;
END_VAR
Check.IsTrue(ipContainer.IsValid, 'ipContainer must be a valid container');
Check.IsTrue(ipContainer.IsType(TC_GLOBAL_CONST_LIST.ContainerType_Vector_TcVnVector2_UINT), 'ipContainer contains incorrect type');
END_METHOD

END_FUNCTION_BLOCK

// Nodes/Container Statistics/MaxElementwise/Node_F_VN_MaxElementElementwise_TcVnVector2_USINT
{attribute 'linkalways'} 
{attribute 'no_explicit_call' := 'This FB is a CLASS and must be accessed using methods or properties'}
{attribute 'enable_dynamic_creation'}
FUNCTION_BLOCK Node_F_VN_MaxElementElementwise_TcVnVector2_USINT EXTENDS VisionNode
VAR
    ipContainer : _ITcVnContainer;
    aMax : _TcVnVector2_USINT;
    hrPrev : _HRESULT(S_OK);
    hresult : _HRESULT(S_OK);
END_VAR

METHOD FB_init : BOOL
VAR_INPUT
	bInitRetains : BOOL; // if TRUE, the retain variables are initialized (warm start / cold start)
	bInCopyCode : BOOL;  // if TRUE, the instance afterwards gets moved into the copy code (online change)
END_VAR
AddInput('ipContainer', ipContainer);
AddInput('hrPrev', hrPrev);
AddOutput('ipContainer', ipContainer);
AddOutput('aMax', aMax);
AddOutput('hresult',hresult);
END_METHOD

METHOD PUBLIC  Clone : I_Node
VAR
	pNode : POINTER TO Node_F_VN_MaxElementElementwise_TcVnVector2_USINT;
END_VAR
pNode := __NEW(Node_F_VN_MaxElementElementwise_TcVnVector2_USINT);
Clone := pNode^;
END_METHOD

METHOD PROTECTED OnExecute
hresult.Value := F_VN_MaxElementElementwise_TcVnVector2_USINT(
    ipContainer := ipContainer.Value,
    aMax := aMax.Value,
    hrPrev:= hrPrev.Value);
END_METHOD

METHOD PUBLIC PreExecutionCheck
VAR_INPUT
	Check : I_PreExecutionChecks;
END_VAR
Check.IsTrue(ipContainer.IsValid, 'ipContainer must be a valid container');
Check.IsTrue(ipContainer.IsType(TC_GLOBAL_CONST_LIST.ContainerType_Vector_TcVnVector2_USINT), 'ipContainer contains incorrect type');
END_METHOD

END_FUNCTION_BLOCK

// Nodes/Container Statistics/MaxElementwise/Node_F_VN_MaxElementElementwise_TcVnVector3_INT
{attribute 'linkalways'} 
{attribute 'no_explicit_call' := 'This FB is a CLASS and must be accessed using methods or properties'}
{attribute 'enable_dynamic_creation'}
FUNCTION_BLOCK Node_F_VN_MaxElementElementwise_TcVnVector3_INT EXTENDS VisionNode
VAR
    ipContainer : _ITcVnContainer;
    aMax : _TcVnVector3_INT;
    hrPrev : _HRESULT(S_OK);
    hresult : _HRESULT(S_OK);
END_VAR

METHOD FB_init : BOOL
VAR_INPUT
	bInitRetains : BOOL; // if TRUE, the retain variables are initialized (warm start / cold start)
	bInCopyCode : BOOL;  // if TRUE, the instance afterwards gets moved into the copy code (online change)
END_VAR
AddInput('ipContainer', ipContainer);
AddInput('hrPrev', hrPrev);
AddOutput('ipContainer', ipContainer);
AddOutput('aMax', aMax);
AddOutput('hresult',hresult);
END_METHOD

METHOD PUBLIC  Clone : I_Node
VAR
	pNode : POINTER TO Node_F_VN_MaxElementElementwise_TcVnVector3_INT;
END_VAR
pNode := __NEW(Node_F_VN_MaxElementElementwise_TcVnVector3_INT);
Clone := pNode^;
END_METHOD

METHOD PROTECTED OnExecute
hresult.Value := F_VN_MaxElementElementwise_TcVnVector3_INT(
    ipContainer := ipContainer.Value,
    aMax := aMax.Value,
    hrPrev:= hrPrev.Value);
END_METHOD

METHOD PUBLIC PreExecutionCheck
VAR_INPUT
	Check : I_PreExecutionChecks;
END_VAR
Check.IsTrue(ipContainer.IsValid, 'ipContainer must be a valid container');
Check.IsTrue(ipContainer.IsType(TC_GLOBAL_CONST_LIST.ContainerType_Vector_TcVnVector3_INT), 'ipContainer contains incorrect type');
END_METHOD

END_FUNCTION_BLOCK

// Nodes/Container Statistics/MaxElementwise/Node_F_VN_MaxElementElementwise_TcVnVector3_REAL
{attribute 'linkalways'} 
{attribute 'no_explicit_call' := 'This FB is a CLASS and must be accessed using methods or properties'}
{attribute 'enable_dynamic_creation'}
FUNCTION_BLOCK Node_F_VN_MaxElementElementwise_TcVnVector3_REAL EXTENDS VisionNode
VAR
    ipContainer : _ITcVnContainer;
    aMax : _TcVnVector3_REAL;
    hrPrev : _HRESULT(S_OK);
    hresult : _HRESULT(S_OK);
END_VAR

METHOD FB_init : BOOL
VAR_INPUT
	bInitRetains : BOOL; // if TRUE, the retain variables are initialized (warm start / cold start)
	bInCopyCode : BOOL;  // if TRUE, the instance afterwards gets moved into the copy code (online change)
END_VAR
AddInput('ipContainer', ipContainer);
AddInput('hrPrev', hrPrev);
AddOutput('ipContainer', ipContainer);
AddOutput('aMax', aMax);
AddOutput('hresult',hresult);
END_METHOD

METHOD PUBLIC  Clone : I_Node
VAR
	pNode : POINTER TO Node_F_VN_MaxElementElementwise_TcVnVector3_REAL;
END_VAR
pNode := __NEW(Node_F_VN_MaxElementElementwise_TcVnVector3_REAL);
Clone := pNode^;
END_METHOD

METHOD PROTECTED OnExecute
hresult.Value := F_VN_MaxElementElementwise_TcVnVector3_REAL(
    ipContainer := ipContainer.Value,
    aMax := aMax.Value,
    hrPrev:= hrPrev.Value);
END_METHOD

METHOD PUBLIC PreExecutionCheck
VAR_INPUT
	Check : I_PreExecutionChecks;
END_VAR
Check.IsTrue(ipContainer.IsValid, 'ipContainer must be a valid container');
Check.IsTrue(ipContainer.IsType(TC_GLOBAL_CONST_LIST.ContainerType_Vector_TcVnVector3_REAL), 'ipContainer contains incorrect type');
END_METHOD

END_FUNCTION_BLOCK

// Nodes/Container Statistics/MaxElementwise/Node_F_VN_MaxElementElementwise_TcVnVector3_SINT
{attribute 'linkalways'} 
{attribute 'no_explicit_call' := 'This FB is a CLASS and must be accessed using methods or properties'}
{attribute 'enable_dynamic_creation'}
FUNCTION_BLOCK Node_F_VN_MaxElementElementwise_TcVnVector3_SINT EXTENDS VisionNode
VAR
    ipContainer : _ITcVnContainer;
    aMax : _TcVnVector3_SINT;
    hrPrev : _HRESULT(S_OK);
    hresult : _HRESULT(S_OK);
END_VAR

METHOD FB_init : BOOL
VAR_INPUT
	bInitRetains : BOOL; // if TRUE, the retain variables are initialized (warm start / cold start)
	bInCopyCode : BOOL;  // if TRUE, the instance afterwards gets moved into the copy code (online change)
END_VAR
AddInput('ipContainer', ipContainer);
AddInput('hrPrev', hrPrev);
AddOutput('ipContainer', ipContainer);
AddOutput('aMax', aMax);
AddOutput('hresult',hresult);
END_METHOD

METHOD PUBLIC  Clone : I_Node
VAR
	pNode : POINTER TO Node_F_VN_MaxElementElementwise_TcVnVector3_SINT;
END_VAR
pNode := __NEW(Node_F_VN_MaxElementElementwise_TcVnVector3_SINT);
Clone := pNode^;
END_METHOD

METHOD PROTECTED OnExecute
hresult.Value := F_VN_MaxElementElementwise_TcVnVector3_SINT(
    ipContainer := ipContainer.Value,
    aMax := aMax.Value,
    hrPrev:= hrPrev.Value);
END_METHOD

METHOD PUBLIC PreExecutionCheck
VAR_INPUT
	Check : I_PreExecutionChecks;
END_VAR
Check.IsTrue(ipContainer.IsValid, 'ipContainer must be a valid container');
Check.IsTrue(ipContainer.IsType(TC_GLOBAL_CONST_LIST.ContainerType_Vector_TcVnVector3_SINT), 'ipContainer contains incorrect type');
END_METHOD

END_FUNCTION_BLOCK

// Nodes/Container Statistics/MaxElementwise/Node_F_VN_MaxElementElementwise_TcVnVector3_UINT
{attribute 'linkalways'} 
{attribute 'no_explicit_call' := 'This FB is a CLASS and must be accessed using methods or properties'}
{attribute 'enable_dynamic_creation'}
FUNCTION_BLOCK Node_F_VN_MaxElementElementwise_TcVnVector3_UINT EXTENDS VisionNode
VAR
    ipContainer : _ITcVnContainer;
    aMax : _TcVnVector3_UINT;
    hrPrev : _HRESULT(S_OK);
    hresult : _HRESULT(S_OK);
END_VAR

METHOD FB_init : BOOL
VAR_INPUT
	bInitRetains : BOOL; // if TRUE, the retain variables are initialized (warm start / cold start)
	bInCopyCode : BOOL;  // if TRUE, the instance afterwards gets moved into the copy code (online change)
END_VAR
AddInput('ipContainer', ipContainer);
AddInput('hrPrev', hrPrev);
AddOutput('ipContainer', ipContainer);
AddOutput('aMax', aMax);
AddOutput('hresult',hresult);
END_METHOD

METHOD PUBLIC  Clone : I_Node
VAR
	pNode : POINTER TO Node_F_VN_MaxElementElementwise_TcVnVector3_UINT;
END_VAR
pNode := __NEW(Node_F_VN_MaxElementElementwise_TcVnVector3_UINT);
Clone := pNode^;
END_METHOD

METHOD PROTECTED OnExecute
hresult.Value := F_VN_MaxElementElementwise_TcVnVector3_UINT(
    ipContainer := ipContainer.Value,
    aMax := aMax.Value,
    hrPrev:= hrPrev.Value);
END_METHOD

METHOD PUBLIC PreExecutionCheck
VAR_INPUT
	Check : I_PreExecutionChecks;
END_VAR
Check.IsTrue(ipContainer.IsValid, 'ipContainer must be a valid container');
Check.IsTrue(ipContainer.IsType(TC_GLOBAL_CONST_LIST.ContainerType_Vector_TcVnVector3_UINT), 'ipContainer contains incorrect type');
END_METHOD

END_FUNCTION_BLOCK

// Nodes/Container Statistics/MaxElementwise/Node_F_VN_MaxElementElementwise_TcVnVector3_USINT
{attribute 'linkalways'} 
{attribute 'no_explicit_call' := 'This FB is a CLASS and must be accessed using methods or properties'}
{attribute 'enable_dynamic_creation'}
FUNCTION_BLOCK Node_F_VN_MaxElementElementwise_TcVnVector3_USINT EXTENDS VisionNode
VAR
    ipContainer : _ITcVnContainer;
    aMax : _TcVnVector3_USINT;
    hrPrev : _HRESULT(S_OK);
    hresult : _HRESULT(S_OK);
END_VAR

METHOD FB_init : BOOL
VAR_INPUT
	bInitRetains : BOOL; // if TRUE, the retain variables are initialized (warm start / cold start)
	bInCopyCode : BOOL;  // if TRUE, the instance afterwards gets moved into the copy code (online change)
END_VAR
AddInput('ipContainer', ipContainer);
AddInput('hrPrev', hrPrev);
AddOutput('ipContainer', ipContainer);
AddOutput('aMax', aMax);
AddOutput('hresult',hresult);
END_METHOD

METHOD PUBLIC  Clone : I_Node
VAR
	pNode : POINTER TO Node_F_VN_MaxElementElementwise_TcVnVector3_USINT;
END_VAR
pNode := __NEW(Node_F_VN_MaxElementElementwise_TcVnVector3_USINT);
Clone := pNode^;
END_METHOD

METHOD PROTECTED OnExecute
hresult.Value := F_VN_MaxElementElementwise_TcVnVector3_USINT(
    ipContainer := ipContainer.Value,
    aMax := aMax.Value,
    hrPrev:= hrPrev.Value);
END_METHOD

METHOD PUBLIC PreExecutionCheck
VAR_INPUT
	Check : I_PreExecutionChecks;
END_VAR
Check.IsTrue(ipContainer.IsValid, 'ipContainer must be a valid container');
Check.IsTrue(ipContainer.IsType(TC_GLOBAL_CONST_LIST.ContainerType_Vector_TcVnVector3_USINT), 'ipContainer contains incorrect type');
END_METHOD

END_FUNCTION_BLOCK

// Nodes/Container Statistics/MaxElementwise/Node_F_VN_MaxElementElementwise_TcVnVector4_DINT
{attribute 'linkalways'} 
{attribute 'no_explicit_call' := 'This FB is a CLASS and must be accessed using methods or properties'}
{attribute 'enable_dynamic_creation'}
FUNCTION_BLOCK Node_F_VN_MaxElementElementwise_TcVnVector4_DINT EXTENDS VisionNode
VAR
    ipContainer : _ITcVnContainer;
    aMax : _TcVnVector4_DINT;
    hrPrev : _HRESULT(S_OK);
    hresult : _HRESULT(S_OK);
END_VAR

METHOD FB_init : BOOL
VAR_INPUT
	bInitRetains : BOOL; // if TRUE, the retain variables are initialized (warm start / cold start)
	bInCopyCode : BOOL;  // if TRUE, the instance afterwards gets moved into the copy code (online change)
END_VAR
AddInput('ipContainer', ipContainer);
AddInput('hrPrev', hrPrev);
AddOutput('ipContainer', ipContainer);
AddOutput('aMax', aMax);
AddOutput('hresult',hresult);
END_METHOD

METHOD PUBLIC  Clone : I_Node
VAR
	pNode : POINTER TO Node_F_VN_MaxElementElementwise_TcVnVector4_DINT;
END_VAR
pNode := __NEW(Node_F_VN_MaxElementElementwise_TcVnVector4_DINT);
Clone := pNode^;
END_METHOD

METHOD PROTECTED OnExecute
hresult.Value := F_VN_MaxElementElementwise_TcVnVector4_DINT(
    ipContainer := ipContainer.Value,
    aMax := aMax.Value,
    hrPrev:= hrPrev.Value);
END_METHOD

METHOD PUBLIC PreExecutionCheck
VAR_INPUT
	Check : I_PreExecutionChecks;
END_VAR
Check.IsTrue(ipContainer.IsValid, 'ipContainer must be a valid container');
Check.IsTrue(ipContainer.IsType(TC_GLOBAL_CONST_LIST.ContainerType_Vector_TcVnVector4_DINT), 'ipContainer contains incorrect type');
END_METHOD

END_FUNCTION_BLOCK

// Nodes/Container Statistics/MaxElementwise/Node_F_VN_MaxElementElementwise_TcVnVector4_INT
{attribute 'linkalways'} 
{attribute 'no_explicit_call' := 'This FB is a CLASS and must be accessed using methods or properties'}
{attribute 'enable_dynamic_creation'}
FUNCTION_BLOCK Node_F_VN_MaxElementElementwise_TcVnVector4_INT EXTENDS VisionNode
VAR
    ipContainer : _ITcVnContainer;
    aMax : _TcVnVector4_INT;
    hrPrev : _HRESULT(S_OK);
    hresult : _HRESULT(S_OK);
END_VAR

METHOD FB_init : BOOL
VAR_INPUT
	bInitRetains : BOOL; // if TRUE, the retain variables are initialized (warm start / cold start)
	bInCopyCode : BOOL;  // if TRUE, the instance afterwards gets moved into the copy code (online change)
END_VAR
AddInput('ipContainer', ipContainer);
AddInput('hrPrev', hrPrev);
AddOutput('ipContainer', ipContainer);
AddOutput('aMax', aMax);
AddOutput('hresult',hresult);
END_METHOD

METHOD PUBLIC  Clone : I_Node
VAR
	pNode : POINTER TO Node_F_VN_MaxElementElementwise_TcVnVector4_INT;
END_VAR
pNode := __NEW(Node_F_VN_MaxElementElementwise_TcVnVector4_INT);
Clone := pNode^;
END_METHOD

METHOD PROTECTED OnExecute
hresult.Value := F_VN_MaxElementElementwise_TcVnVector4_INT(
    ipContainer := ipContainer.Value,
    aMax := aMax.Value,
    hrPrev:= hrPrev.Value);
END_METHOD

METHOD PUBLIC PreExecutionCheck
VAR_INPUT
	Check : I_PreExecutionChecks;
END_VAR
Check.IsTrue(ipContainer.IsValid, 'ipContainer must be a valid container');
Check.IsTrue(ipContainer.IsType(TC_GLOBAL_CONST_LIST.ContainerType_Vector_TcVnVector4_INT), 'ipContainer contains incorrect type');
END_METHOD

END_FUNCTION_BLOCK

// Nodes/Container Statistics/MaxElementwise/Node_F_VN_MaxElementElementwise_TcVnVector4_LREAL
{attribute 'linkalways'} 
{attribute 'no_explicit_call' := 'This FB is a CLASS and must be accessed using methods or properties'}
{attribute 'enable_dynamic_creation'}
FUNCTION_BLOCK Node_F_VN_MaxElementElementwise_TcVnVector4_LREAL EXTENDS VisionNode
VAR
    ipContainer : _ITcVnContainer;
    aMax : _TcVnVector4_LREAL;
    hrPrev : _HRESULT(S_OK);
    hresult : _HRESULT(S_OK);
END_VAR

METHOD FB_init : BOOL
VAR_INPUT
	bInitRetains : BOOL; // if TRUE, the retain variables are initialized (warm start / cold start)
	bInCopyCode : BOOL;  // if TRUE, the instance afterwards gets moved into the copy code (online change)
END_VAR
AddInput('ipContainer', ipContainer);
AddInput('hrPrev', hrPrev);
AddOutput('ipContainer', ipContainer);
AddOutput('aMax', aMax);
AddOutput('hresult',hresult);
END_METHOD

METHOD PUBLIC  Clone : I_Node
VAR
	pNode : POINTER TO Node_F_VN_MaxElementElementwise_TcVnVector4_LREAL;
END_VAR
pNode := __NEW(Node_F_VN_MaxElementElementwise_TcVnVector4_LREAL);
Clone := pNode^;
END_METHOD

METHOD PROTECTED OnExecute
hresult.Value := F_VN_MaxElementElementwise_TcVnVector4_LREAL(
    ipContainer := ipContainer.Value,
    aMax := aMax.Value,
    hrPrev:= hrPrev.Value);
END_METHOD

METHOD PUBLIC PreExecutionCheck
VAR_INPUT
	Check : I_PreExecutionChecks;
END_VAR
Check.IsTrue(ipContainer.IsValid, 'ipContainer must be a valid container');
Check.IsTrue(ipContainer.IsType(TC_GLOBAL_CONST_LIST.ContainerType_Vector_TcVnVector4_LREAL), 'ipContainer contains incorrect type');
END_METHOD

END_FUNCTION_BLOCK

// Nodes/Container Statistics/MaxElementwise/Node_F_VN_MaxElementElementwise_TcVnVector4_REAL
{attribute 'linkalways'} 
{attribute 'no_explicit_call' := 'This FB is a CLASS and must be accessed using methods or properties'}
{attribute 'enable_dynamic_creation'}
FUNCTION_BLOCK Node_F_VN_MaxElementElementwise_TcVnVector4_REAL EXTENDS VisionNode
VAR
    ipContainer : _ITcVnContainer;
    aMax : _TcVnVector4_REAL;
    hrPrev : _HRESULT(S_OK);
    hresult : _HRESULT(S_OK);
END_VAR

METHOD FB_init : BOOL
VAR_INPUT
	bInitRetains : BOOL; // if TRUE, the retain variables are initialized (warm start / cold start)
	bInCopyCode : BOOL;  // if TRUE, the instance afterwards gets moved into the copy code (online change)
END_VAR
AddInput('ipContainer', ipContainer);
AddInput('hrPrev', hrPrev);
AddOutput('ipContainer', ipContainer);
AddOutput('aMax', aMax);
AddOutput('hresult',hresult);
END_METHOD

METHOD PUBLIC  Clone : I_Node
VAR
	pNode : POINTER TO Node_F_VN_MaxElementElementwise_TcVnVector4_REAL;
END_VAR
pNode := __NEW(Node_F_VN_MaxElementElementwise_TcVnVector4_REAL);
Clone := pNode^;
END_METHOD

METHOD PROTECTED OnExecute
hresult.Value := F_VN_MaxElementElementwise_TcVnVector4_REAL(
    ipContainer := ipContainer.Value,
    aMax := aMax.Value,
    hrPrev:= hrPrev.Value);
END_METHOD

METHOD PUBLIC PreExecutionCheck
VAR_INPUT
	Check : I_PreExecutionChecks;
END_VAR
Check.IsTrue(ipContainer.IsValid, 'ipContainer must be a valid container');
Check.IsTrue(ipContainer.IsType(TC_GLOBAL_CONST_LIST.ContainerType_Vector_TcVnVector4_REAL), 'ipContainer contains incorrect type');
END_METHOD

END_FUNCTION_BLOCK

// Nodes/Container Statistics/MaxElementwise/Node_F_VN_MaxElementElementwise_TcVnVector4_SINT
{attribute 'linkalways'} 
{attribute 'no_explicit_call' := 'This FB is a CLASS and must be accessed using methods or properties'}
{attribute 'enable_dynamic_creation'}
FUNCTION_BLOCK Node_F_VN_MaxElementElementwise_TcVnVector4_SINT EXTENDS VisionNode
VAR
    ipContainer : _ITcVnContainer;
    aMax : _TcVnVector4_SINT;
    hrPrev : _HRESULT(S_OK);
    hresult : _HRESULT(S_OK);
END_VAR

METHOD FB_init : BOOL
VAR_INPUT
	bInitRetains : BOOL; // if TRUE, the retain variables are initialized (warm start / cold start)
	bInCopyCode : BOOL;  // if TRUE, the instance afterwards gets moved into the copy code (online change)
END_VAR
AddInput('ipContainer', ipContainer);
AddInput('hrPrev', hrPrev);
AddOutput('ipContainer', ipContainer);
AddOutput('aMax', aMax);
AddOutput('hresult',hresult);
END_METHOD

METHOD PUBLIC  Clone : I_Node
VAR
	pNode : POINTER TO Node_F_VN_MaxElementElementwise_TcVnVector4_SINT;
END_VAR
pNode := __NEW(Node_F_VN_MaxElementElementwise_TcVnVector4_SINT);
Clone := pNode^;
END_METHOD

METHOD PROTECTED OnExecute
hresult.Value := F_VN_MaxElementElementwise_TcVnVector4_SINT(
    ipContainer := ipContainer.Value,
    aMax := aMax.Value,
    hrPrev:= hrPrev.Value);
END_METHOD

METHOD PUBLIC PreExecutionCheck
VAR_INPUT
	Check : I_PreExecutionChecks;
END_VAR
Check.IsTrue(ipContainer.IsValid, 'ipContainer must be a valid container');
Check.IsTrue(ipContainer.IsType(TC_GLOBAL_CONST_LIST.ContainerType_Vector_TcVnVector4_SINT), 'ipContainer contains incorrect type');
END_METHOD

END_FUNCTION_BLOCK

